LIN {X 0,Y 199.613,Z 290.431,A -85,B 0,C 180,E1 -21475.713,E2 -21475.713} C_VEL
LIN {X 0,Y 199.653,Z 290.436,A -85,B 0,C 180,E1 -21477.571,E2 -21477.571} C_VEL
LIN {X 0,Y 200.584,Z 293.129,A -85,B 0,C 180,E1 -21477.855,E2 -21477.855} C_VEL
LIN {X 0,Y 203.702,Z 298.377,A -85,B 0,C 180,E1 -21478.627,E2 -21478.627} C_VEL
LIN {X 0,Y 211.896,Z 314.5,A -85,B 0,C 180,E1 -21480.608,E2 -21480.608} C_VEL
LIN {X 0,Y 215.116,Z 321.856,A -85,B 0,C 180,E1 -21481.374,E2 -21481.374} C_VEL
LIN {X 0,Y 213.786,Z 358.585,A -85,B 0,C 180,E1 -21482.597,E2 -21482.597} C_VEL
LIN {X 0,Y 213.285,Z 367.836,A -85,B 0,C 180,E1 -21483.118,E2 -21483.118} C_VEL
LIN {X 0,Y 212.677,Z 375.597,A -85,B 0,C 180,E1 -21483.748,E2 -21483.748} C_VEL
LIN {X 0,Y 211.647,Z 384.419,A -85,B 0,C 180,E1 -21484.688,E2 -21484.688} C_VEL
LIN {X 0,Y 210.204,Z 392.837,A -85,B 0,C 180,E1 -21485.821,E2 -21485.821} C_VEL
LIN {X 0,Y 208.91,Z 399.701,A -85,B 0,C 180,E1 -21486.977,E2 -21486.977} C_VEL
LIN {X 0,Y 207.269,Z 407.588,A -85,B 0,C 180,E1 -21488.622,E2 -21488.622} C_VEL
LIN {X 0,Y 205.97,Z 413.247,A -85,B 0,C 180,E1 -21490.048,E2 -21490.048} C_VEL
LIN {X 0,Y 204.385,Z 419.566,A -85,B 0,C 180,E1 -21491.971,E2 -21491.971} C_VEL
LIN {X 0,Y 202.851,Z 424.822,A -85,B 0,C 180,E1 -21493.908,E2 -21493.908} C_VEL
LIN {X 0,Y 201.567,Z 429.206,A -85,B 0,C 180,E1 -21495.872,E2 -21495.872} C_VEL
LIN {X 0,Y 200.108,Z 434.351,A -85,B 0,C 180,E1 -21498.861,E2 -21498.861} C_VEL
LIN {X 0,Y 199.427,Z 436.755,A -85,B 0,C 180,E1 -21500.664,E2 -21500.664} C_VEL
LIN {X 0,Y 198.499,Z 439.877,A -85,B 0,C 180,E1 -21503.902,E2 -21503.902} C_VEL
LIN {X 0,Y 198.087,Z 441.139,A -85,B 0,C 180,E1 -21505.93,E2 -21505.93} C_VEL
LIN {X 0,Y 197.808,Z 441.935,A -85,B 0,C 180,E1 -21507.963,E2 -21507.963} C_VEL
LIN {X 0,Y 197.72,Z 442.238,A -85,B 0,C 180,E1 -21509.999,E2 -21509.999} C_VEL
LIN {X 0,Y 197.805,Z 441.958,A -85,B 0,C 180,E1 -21512.035,E2 -21512.035} C_VEL
LIN {X 0,Y 198.078,Z 441.21,A -85,B 0,C 180,E1 -21514.068,E2 -21514.068} C_VEL
LIN {X 0,Y 198.49,Z 439.996,A -85,B 0,C 180,E1 -21516.096,E2 -21516.096} C_VEL
LIN {X 0,Y 199.036,Z 438.296,A -85,B 0,C 180,E1 -21518.119,E2 -21518.119} C_VEL
LIN {X 0,Y 200.093,Z 434.572,A -85,B 0,C 180,E1 -21521.137,E2 -21521.137} C_VEL
LIN {X 0,Y 201.547,Z 429.487,A -85,B 0,C 180,E1 -21524.127,E2 -21524.127} C_VEL
LIN {X 0,Y 203.159,Z 424.005,A -85,B 0,C 180,E1 -21526.581,E2 -21526.581} C_VEL
LIN {X 0,Y 205.084,Z 417.109,A -85,B 0,C 180,E1 -21528.998,E2 -21528.998} C_VEL
LIN {X 0,Y 206.999,Z 409.189,A -85,B 0,C 180,E1 -21531.144,E2 -21531.144} C_VEL
LIN {X 0,Y 208.645,Z 401.633,A -85,B 0,C 180,E1 -21532.79,E2 -21532.79} C_VEL
LIN {X 0,Y 210.207,Z 393.703,A -85,B 0,C 180,E1 -21534.176,E2 -21534.176} C_VEL
LIN {X 0,Y 211.587,Z 385.502,A -85,B 0,C 180,E1 -21535.317,E2 -21535.317} C_VEL
LIN {X 0,Y 212.67,Z 377.081,A -85,B 0,C 180,E1 -21536.241,E2 -21536.241} C_VEL
LIN {X 0,Y 213.409,Z 367.929,A -85,B 0,C 180,E1 -21537.009,E2 -21537.009} C_VEL
LIN {X 0,Y 213.899,Z 358.992,A -85,B 0,C 180,E1 -21537.518,E2 -21537.518} C_VEL
LIN {X 0,Y 215.253,Z 322.206,A -85,B 0,C 180,E1 -21538.745,E2 -21538.745} C_VEL
LIN {X 0,Y 209.18,Z 308.863,A -85,B 0,C 180,E1 -21540.195,E2 -21540.195} C_VEL
LIN {X 0,Y 201.446,Z 294.316,A -85,B 0,C 180,E1 -21542.103,E2 -21542.103} C_VEL
LIN {X 0,Y 199.955,Z 291.746,A -85,B 0,C 180,E1 -21542.483,E2 -21542.483} C_VEL
LIN {X 0,Y 199.655,Z 290.429,A -85,B 0,C 180,E1 -21542.638,E2 -21542.638} C_VEL
LIN {X 0,Y 199.613,Z 290.425,A -85,B 0,C 180,E1 -21546.764,E2 -21546.764} C_VEL
LIN {X 0,Y 199.591,Z 290.435,A -85,B 0,C 180,E1 -21549.331,E2 -21549.331} C_VEL
LIN {X 0,Y 199.562,Z 290.428,A -85,B 0,C 180,E1 -21552.306,E2 -21552.306} C_VEL
LIN {X 0,Y 199.573,Z 290.436,A -85,B 0,C 180,E1 -21555.226,E2 -21555.226} C_VEL
LIN {X 0,Y 199.566,Z 290.42,A -85,B 0,C 180,E1 -21558.001,E2 -21558.001} C_VEL
LIN {X 0,Y 199.593,Z 290.431,A -85,B 0,C 180,E1 -21560.772,E2 -21560.772} C_VEL
LIN {X 0,Y 199.607,Z 290.432,A -85,B 0,C 180,E1 -21565.712,E2 -21565.712} C_VEL
LIN {X 0,Y 199.682,Z 290.419,A -85,B 0,C 180,E1 -21568.133,E2 -21568.133} C_VEL
LIN {X 0,Y 199.638,Z 290.422,A -85,B 0,C 180,E1 -21572.764,E2 -21572.764} C_VEL
LIN {X 0,Y 199.674,Z 290.421,A -85,B 0,C 180,E1 -21577.221,E2 -21577.221} C_VEL
LIN {X 0,Y 199.742,Z 290.411,A -85,B 0,C 180,E1 -21581.802,E2 -21581.802} C_VEL
LIN {X 0,Y 199.766,Z 290.389,A -85,B 0,C 180,E1 -21585.743,E2 -21585.743} C_VEL
LIN {X 0,Y 200.019,Z 290.381,A -85,B 0,C 180,E1 -21589.881,E2 -21589.881} C_VEL
LIN {X 0,Y 199.994,Z 290.372,A -85,B 0,C 180,E1 -21593.948,E2 -21593.948} C_VEL
LIN {X 0,Y 200.28,Z 290.332,A -85,B 0,C 180,E1 -21597.989,E2 -21597.989} C_VEL
LIN {X 0,Y 200.442,Z 290.324,A -85,B 0,C 180,E1 -21600,E2 -21600} C_VEL
LIN {X 0,Y 199.983,Z 290.383,A -85,B 0,C 180,E1 -21604.03,E2 -21604.03} C_VEL
LIN {X 0,Y 200.07,Z 290.377,A -85,B 0,C 180,E1 -21608.077,E2 -21608.077} C_VEL
LIN {X 0,Y 199.848,Z 290.402,A -85,B 0,C 180,E1 -21612.181,E2 -21612.181} C_VEL
LIN {X 0,Y 199.738,Z 290.415,A -85,B 0,C 180,E1 -21616.349,E2 -21616.349} C_VEL
LIN {X 0,Y 199.639,Z 290.427,A -85,B 0,C 180,E1 -21620.612,E2 -21620.612} C_VEL
LIN {X 0,Y 199.621,Z 290.428,A -85,B 0,C 180,E1 -21624.991,E2 -21624.991} C_VEL
LIN {X 0,Y 199.602,Z 290.437,A -85,B 0,C 180,E1 -21629.534,E2 -21629.534} C_VEL
LIN {X 0,Y 199.661,Z 290.429,A -85,B 0,C 180,E1 -21632.353,E2 -21632.353} C_VEL
LIN {X 0,Y 199.611,Z 290.436,A -85,B 0,C 180,E1 -21636.765,E2 -21636.765} C_VEL
LIN {X 0,Y 199.59,Z 290.44,A -85,B 0,C 180,E1 -21639.332,E2 -21639.332} C_VEL
LIN {X 0,Y 199.561,Z 290.441,A -85,B 0,C 180,E1 -21642.308,E2 -21642.308} C_VEL
LIN {X 0,Y 199.572,Z 290.441,A -85,B 0,C 180,E1 -21645.228,E2 -21645.228} C_VEL
LIN {X 0,Y 199.566,Z 290.44,A -85,B 0,C 180,E1 -21648.003,E2 -21648.003} C_VEL
LIN {X 0,Y 199.653,Z 290.544,A -85,B 0,C 180,E1 -21651.413,E2 -21651.413} C_VEL
LIN {X 0,Y 201.4,Z 297.896,A -85,B 0,C 180,E1 -21655.456,E2 -21655.456} C_VEL
LIN {X 0,Y 202.273,Z 302.073,A -85,B 0,C 180,E1 -21657.631,E2 -21657.631} C_VEL
LIN {X 0,Y 208.961,Z 318.344,A -85,B 0,C 180,E1 -21659.408,E2 -21659.408} C_VEL
LIN {X 0,Y 210.715,Z 328.85,A -85,B 0,C 180,E1 -21660.089,E2 -21660.089} C_VEL
LIN {X 0,Y 211.052,Z 334.648,A -85,B 0,C 180,E1 -21660.363,E2 -21660.363} C_VEL
LIN {X 0,Y 209.97,Z 344.437,A -85,B 0,C 180,E1 -21660.573,E2 -21660.573} C_VEL
LIN {X 0,Y 208.579,Z 352.327,A -85,B 0,C 180,E1 -21660.665,E2 -21660.665} C_VEL
LIN {X 0,Y 207.672,Z 360.248,A -85,B 0,C 180,E1 -21660.833,E2 -21660.833} C_VEL
LIN {X 0,Y 206.792,Z 381.239,A -85,B 0,C 180,E1 -21661.59,E2 -21661.59} C_VEL
LIN {X 0,Y 205.784,Z 392.316,A -85,B 0,C 180,E1 -21662.27,E2 -21662.27} C_VEL
LIN {X 0,Y 204.008,Z 403.947,A -85,B 0,C 180,E1 -21663.396,E2 -21663.396} C_VEL
LIN {X 0,Y 202.279,Z 413.34,A -85,B 0,C 180,E1 -21664.666,E2 -21664.666} C_VEL
LIN {X 0,Y 200.62,Z 420.935,A -85,B 0,C 180,E1 -21665.97,E2 -21665.97} C_VEL
LIN {X 0,Y 198.696,Z 428.802,A -85,B 0,C 180,E1 -21667.653,E2 -21667.653} C_VEL
LIN {X 0,Y 196.738,Z 436.167,A -85,B 0,C 180,E1 -21669.618,E2 -21669.618} C_VEL
LIN {X 0,Y 194.702,Z 443.648,A -85,B 0,C 180,E1 -21672.134,E2 -21672.134} C_VEL
LIN {X 0,Y 192.709,Z 450.484,A -85,B 0,C 180,E1 -21675.211,E2 -21675.211} C_VEL
LIN {X 0,Y 191.391,Z 455.696,A -85,B 0,C 180,E1 -21678.349,E2 -21678.349} C_VEL
LIN {X 0,Y 190.642,Z 459.536,A -85,B 0,C 180,E1 -21681.521,E2 -21681.521} C_VEL
LIN {X 0,Y 190.376,Z 461.305,A -85,B 0,C 180,E1 -21683.643,E2 -21683.643} C_VEL
LIN {X 0,Y 190.315,Z 462.576,A -85,B 0,C 180,E1 -21685.766,E2 -21685.766} C_VEL
LIN {X 0,Y 190.441,Z 463.373,A -85,B 0,C 180,E1 -21687.886,E2 -21687.886} C_VEL
LIN {X 0,Y 190.608,Z 463.679,A -85,B 0,C 180,E1 -21690.001,E2 -21690.001} C_VEL
LIN {X 0,Y 190.444,Z 463.364,A -85,B 0,C 180,E1 -21692.116,E2 -21692.116} C_VEL
LIN {X 0,Y 190.335,Z 462.437,A -85,B 0,C 180,E1 -21694.474,E2 -21694.474} C_VEL
LIN {X 0,Y 190.378,Z 461.256,A -85,B 0,C 180,E1 -21696.36,E2 -21696.36} C_VEL
LIN {X 0,Y 190.856,Z 458.298,A -85,B 0,C 180,E1 -21699.539,E2 -21699.539} C_VEL
LIN {X 0,Y 191.391,Z 455.606,A -85,B 0,C 180,E1 -21701.653,E2 -21701.653} C_VEL
LIN {X 0,Y 192.708,Z 450.367,A -85,B 0,C 180,E1 -21704.792,E2 -21704.792} C_VEL
LIN {X 0,Y 194.692,Z 443.478,A -85,B 0,C 180,E1 -21707.87,E2 -21707.87} C_VEL
LIN {X 0,Y 196.719,Z 435.963,A -85,B 0,C 180,E1 -21710.386,E2 -21710.386} C_VEL
LIN {X 0,Y 198.719,Z 428.564,A -85,B 0,C 180,E1 -21712.347,E2 -21712.347} C_VEL
LIN {X 0,Y 200.645,Z 420.642,A -85,B 0,C 180,E1 -21714.029,E2 -21714.029} C_VEL
LIN {X 0,Y 202.677,Z 410.766,A -85,B 0,C 180,E1 -21715.686,E2 -21715.686} C_VEL
LIN {X 0,Y 204.651,Z 399.203,A -85,B 0,C 180,E1 -21717.067,E2 -21717.067} C_VEL
LIN {X 0,Y 205.966,Z 389.853,A -85,B 0,C 180,E1 -21717.844,E2 -21717.844} C_VEL
LIN {X 0,Y 206.816,Z 379.973,A -85,B 0,C 180,E1 -21718.409,E2 -21718.409} C_VEL
LIN {X 0,Y 207.545,Z 357.654,A -85,B 0,C 180,E1 -21719.221,E2 -21719.221} C_VEL
LIN {X 0,Y 205.525,Z 338.227,A -85,B 0,C 180,E1 -21720.295,E2 -21720.295} C_VEL
LIN {X 0,Y 203.229,Z 321.421,A -85,B 0,C 180,E1 -21721.343,E2 -21721.343} C_VEL
LIN {X 0,Y 197.805,Z 308.229,A -85,B 0,C 180,E1 -21722.844,E2 -21722.844} C_VEL
LIN {X 0,Y 194.959,Z 301.496,A -85,B 0,C 180,E1 -21723.721,E2 -21723.721} C_VEL
LIN {X 0,Y 193.277,Z 294.173,A -85,B 0,C 180,E1 -21727.825,E2 -21727.825} C_VEL
LIN {X 0,Y 192.543,Z 291.315,A -85,B 0,C 180,E1 -21729.562,E2 -21729.562} C_VEL
LIN {X 0,Y 192.488,Z 291.323,A -85,B 0,C 180,E1 -21733.926,E2 -21733.926} C_VEL
LIN {X 0,Y 192.505,Z 291.321,A -85,B 0,C 180,E1 -21738.918,E2 -21738.918} C_VEL
LIN {X 0,Y 192.582,Z 291.31,A -85,B 0,C 180,E1 -21743.405,E2 -21743.405} C_VEL
LIN {X 0,Y 192.607,Z 291.306,A -85,B 0,C 180,E1 -21747.062,E2 -21747.062} C_VEL
LIN {X 0,Y 192.613,Z 291.303,A -85,B 0,C 180,E1 -21751.684,E2 -21751.684} C_VEL
LIN {X 0,Y 192.658,Z 291.298,A -85,B 0,C 180,E1 -21756.343,E2 -21756.343} C_VEL
LIN {X 0,Y 192.697,Z 291.294,A -85,B 0,C 180,E1 -21761.492,E2 -21761.492} C_VEL
LIN {X 0,Y 192.775,Z 291.285,A -85,B 0,C 180,E1 -21767.365,E2 -21767.365} C_VEL
LIN {X 0,Y 193.021,Z 291.223,A -85,B 0,C 180,E1 -21771.626,E2 -21771.626} C_VEL
LIN {X 0,Y 193.229,Z 291.228,A -85,B 0,C 180,E1 -21777.916,E2 -21777.916} C_VEL
LIN {X 0,Y 193.416,Z 291.198,A -85,B 0,C 180,E1 -21780,E2 -21780} C_VEL
LIN {X 0,Y 192.933,Z 291.235,A -85,B 0,C 180,E1 -21784.178,E2 -21784.178} C_VEL
LIN {X 0,Y 193.024,Z 291.251,A -85,B 0,C 180,E1 -21788.375,E2 -21788.375} C_VEL
LIN {X 0,Y 192.778,Z 291.27,A -85,B 0,C 180,E1 -21792.635,E2 -21792.635} C_VEL
LIN {X 0,Y 192.697,Z 291.288,A -85,B 0,C 180,E1 -21798.508,E2 -21798.508} C_VEL
LIN {X 0,Y 192.613,Z 291.3,A -85,B 0,C 180,E1 -21804.188,E2 -21804.188} C_VEL
LIN {X 0,Y 192.603,Z 291.302,A -85,B 0,C 180,E1 -21808.864,E2 -21808.864} C_VEL
LIN {X 0,Y 192.597,Z 291.295,A -85,B 0,C 180,E1 -21813.186,E2 -21813.186} C_VEL
LIN {X 0,Y 192.543,Z 291.314,A -85,B 0,C 180,E1 -21818.354,E2 -21818.354} C_VEL
LIN {X 0,Y 192.485,Z 291.307,A -85,B 0,C 180,E1 -21823.092,E2 -21823.092} C_VEL
LIN {X 0,Y 192.487,Z 291.323,A -85,B 0,C 180,E1 -21826.906,E2 -21826.906} C_VEL
LIN {X 0,Y 192.543,Z 291.267,A -85,B 0,C 180,E1 -21831.645,E2 -21831.645} C_VEL
LIN {X 0,Y 192.602,Z 291.389,A -85,B 0,C 180,E1 -21836.249,E2 -21836.249} C_VEL
LIN {X 0,Y 193.654,Z 294.262,A -85,B 0,C 180,E1 -21836.586,E2 -21836.586} C_VEL
LIN {X 0,Y 195.306,Z 296.896,A -85,B 0,C 180,E1 -21837.023,E2 -21837.023} C_VEL
LIN {X 0,Y 201.653,Z 308.403,A -85,B 0,C 180,E1 -21838.677,E2 -21838.677} C_VEL
LIN {X 0,Y 208.096,Z 321.908,A -85,B 0,C 180,E1 -21840.297,E2 -21840.297} C_VEL
LIN {X 0,Y 208.918,Z 323.896,A -85,B 0,C 180,E1 -21840.505,E2 -21840.505} C_VEL
LIN {X 0,Y 207.509,Z 359.706,A -85,B 0,C 180,E1 -21841.733,E2 -21841.733} C_VEL
LIN {X 0,Y 206.913,Z 368.837,A -85,B 0,C 180,E1 -21842.269,E2 -21842.269} C_VEL
LIN {X 0,Y 206.141,Z 378.024,A -85,B 0,C 180,E1 -21843.079,E2 -21843.079} C_VEL
LIN {X 0,Y 204.99,Z 386.681,A -85,B 0,C 180,E1 -21844.078,E2 -21844.078} C_VEL
LIN {X 0,Y 203.197,Z 396.224,A -85,B 0,C 180,E1 -21845.477,E2 -21845.477} C_VEL
LIN {X 0,Y 201.461,Z 404.915,A -85,B 0,C 180,E1 -21847.163,E2 -21847.163} C_VEL
LIN {X 0,Y 199.341,Z 413.64,A -85,B 0,C 180,E1 -21849.355,E2 -21849.355} C_VEL
LIN {X 0,Y 197.667,Z 419.959,A -85,B 0,C 180,E1 -21851.337,E2 -21851.337} C_VEL
LIN {X 0,Y 196.071,Z 425.215,A -85,B 0,C 180,E1 -21853.335,E2 -21853.335} C_VEL
LIN {X 0,Y 194.71,Z 429.598,A -85,B 0,C 180,E1 -21855.364,E2 -21855.364} C_VEL
LIN {X 0,Y 193.159,Z 434.744,A -85,B 0,C 180,E1 -21858.455,E2 -21858.455} C_VEL
LIN {X 0,Y 192.374,Z 437.381,A -85,B 0,C 180,E1 -21860.538,E2 -21860.538} C_VEL
LIN {X 0,Y 191.458,Z 440.269,A -85,B 0,C 180,E1 -21863.677,E2 -21863.677} C_VEL
LIN {X 0,Y 191.042,Z 441.529,A -85,B 0,C 180,E1 -21865.78,E2 -21865.78} C_VEL
LIN {X 0,Y 190.748,Z 442.325,A -85,B 0,C 180,E1 -21867.887,E2 -21867.887} C_VEL
LIN {X 0,Y 190.655,Z 442.628,A -85,B 0,C 180,E1 -21869.999,E2 -21869.999} C_VEL
LIN {X 0,Y 190.745,Z 442.348,A -85,B 0,C 180,E1 -21872.11,E2 -21872.11} C_VEL
LIN {X 0,Y 191.034,Z 441.599,A -85,B 0,C 180,E1 -21874.218,E2 -21874.218} C_VEL
LIN {X 0,Y 191.449,Z 440.387,A -85,B 0,C 180,E1 -21876.322,E2 -21876.322} C_VEL
LIN {X 0,Y 192.316,Z 437.661,A -85,B 0,C 180,E1 -21879.358,E2 -21879.358} C_VEL
LIN {X 0,Y 193.151,Z 434.962,A -85,B 0,C 180,E1 -21881.543,E2 -21881.543} C_VEL
LIN {X 0,Y 194.69,Z 429.876,A -85,B 0,C 180,E1 -21884.636,E2 -21884.636} C_VEL
LIN {X 0,Y 196.377,Z 424.395,A -85,B 0,C 180,E1 -21887.172,E2 -21887.172} C_VEL
LIN {X 0,Y 198.419,Z 417.496,A -85,B 0,C 180,E1 -21889.662,E2 -21889.662} C_VEL
LIN {X 0,Y 200.402,Z 409.577,A -85,B 0,C 180,E1 -21891.876,E2 -21891.876} C_VEL
LIN {X 0,Y 202.139,Z 402.02,A -85,B 0,C 180,E1 -21893.567,E2 -21893.567} C_VEL
LIN {X 0,Y 203.786,Z 394.088,A -85,B 0,C 180,E1 -21894.989,E2 -21894.989} C_VEL
LIN {X 0,Y 205.222,Z 385.886,A -85,B 0,C 180,E1 -21896.161,E2 -21896.161} C_VEL
LIN {X 0,Y 206.312,Z 377.646,A -85,B 0,C 180,E1 -21897.094,E2 -21897.094} C_VEL
LIN {X 0,Y 207.096,Z 368.746,A -85,B 0,C 180,E1 -21897.866,E2 -21897.866} C_VEL
LIN {X 0,Y 207.647,Z 359.505,A -85,B 0,C 180,E1 -21898.413,E2 -21898.413} C_VEL
LIN {X 0,Y 209.064,Z 324.183,A -85,B 0,C 180,E1 -21899.617,E2 -21899.617} C_VEL
LIN {X 0,Y 202.494,Z 310.086,A -85,B 0,C 180,E1 -21901.269,E2 -21901.269} C_VEL
LIN {X 0,Y 196.233,Z 298.469,A -85,B 0,C 180,E1 -21902.899,E2 -21902.899} C_VEL
LIN {X 0,Y 194.061,Z 294.841,A -85,B 0,C 180,E1 -21903.479,E2 -21903.479} C_VEL
LIN {X 0,Y 192.734,Z 292.117,A -85,B 0,C 180,E1 -21903.864,E2 -21903.864} C_VEL
LIN {X 0,Y 192.573,Z 291.311,A -85,B 0,C 180,E1 -21903.954,E2 -21903.954} C_VEL
LIN {X 0,Y 192.538,Z 291.315,A -85,B 0,C 180,E1 -21908.353,E2 -21908.353} C_VEL
LIN {X 0,Y 192.482,Z 291.316,A -85,B 0,C 180,E1 -21913.092,E2 -21913.092} C_VEL
LIN {X 0,Y 192.481,Z 291.306,A -85,B 0,C 180,E1 -21916.906,E2 -21916.906} C_VEL
LIN {X 0,Y 192.537,Z 291.313,A -85,B 0,C 180,E1 -21921.645,E2 -21921.645} C_VEL
LIN {X 0,Y 192.591,Z 291.303,A -85,B 0,C 180,E1 -21926.812,E2 -21926.812} C_VEL
LIN {X 0,Y 192.616,Z 291.298,A -85,B 0,C 180,E1 -21931.684,E2 -21931.684} C_VEL
LIN {X 0,Y 192.667,Z 291.295,A -85,B 0,C 180,E1 -21936.343,E2 -21936.343} C_VEL
LIN {X 0,Y 192.69,Z 291.291,A -85,B 0,C 180,E1 -21941.491,E2 -21941.491} C_VEL
LIN {X 0,Y 192.77,Z 291.27,A -85,B 0,C 180,E1 -21947.364,E2 -21947.364} C_VEL
LIN {X 0,Y 193.017,Z 291.252,A -85,B 0,C 180,E1 -21951.625,E2 -21951.625} C_VEL
LIN {X 0,Y 193.224,Z 291.208,A -85,B 0,C 180,E1 -21957.915,E2 -21957.915} C_VEL
LIN {X 0,Y 193.409,Z 291.199,A -85,B 0,C 180,E1 -21960,E2 -21960} C_VEL
LIN {X 0,Y 192.93,Z 291.26,A -85,B 0,C 180,E1 -21964.178,E2 -21964.178} C_VEL
LIN {X 0,Y 193.021,Z 291.254,A -85,B 0,C 180,E1 -21968.374,E2 -21968.374} C_VEL
LIN {X 0,Y 192.77,Z 291.286,A -85,B 0,C 180,E1 -21972.635,E2 -21972.635} C_VEL
LIN {X 0,Y 192.69,Z 291.295,A -85,B 0,C 180,E1 -21978.508,E2 -21978.508} C_VEL
LIN {X 0,Y 192.616,Z 291.301,A -85,B 0,C 180,E1 -21984.195,E2 -21984.195} C_VEL
LIN {X 0,Y 192.596,Z 291.309,A -85,B 0,C 180,E1 -21988.865,E2 -21988.865} C_VEL
LIN {X 0,Y 192.59,Z 291.311,A -85,B 0,C 180,E1 -21993.187,E2 -21993.187} C_VEL
LIN {X 0,Y 192.536,Z 291.317,A -85,B 0,C 180,E1 -21998.355,E2 -21998.355} C_VEL
LIN {X 0,Y 192.481,Z 291.325,A -85,B 0,C 180,E1 -22003.094,E2 -22003.094} C_VEL
LIN {X 0,Y 192.481,Z 291.324,A -85,B 0,C 180,E1 -22006.907,E2 -22006.907} C_VEL
LIN {X 0,Y 192.57,Z 291.456,A -85,B 0,C 180,E1 -22010.485,E2 -22010.485} C_VEL
LIN {X 0,Y 194.337,Z 298.658,A -85,B 0,C 180,E1 -22014.648,E2 -22014.648} C_VEL
LIN {X 0,Y 194.997,Z 301.675,A -85,B 0,C 180,E1 -22016.27,E2 -22016.27} C_VEL
LIN {X 0,Y 201.837,Z 317.661,A -85,B 0,C 180,E1 -22018.194,E2 -22018.194} C_VEL
LIN {X 0,Y 203.421,Z 322.25,A -85,B 0,C 180,E1 -22018.652,E2 -22018.652} C_VEL
LIN {X 0,Y 206.196,Z 342.981,A -85,B 0,C 180,E1 -22019.932,E2 -22019.932} C_VEL
LIN {X 0,Y 207.732,Z 358.961,A -85,B 0,C 180,E1 -22020.793,E2 -22020.793} C_VEL
LIN {X 0,Y 207.672,Z 360.248,A -85,B 0,C 180,E1 -22020.833,E2 -22020.833} C_VEL
LIN {X 0,Y 206.824,Z 366.093,A -85,B 0,C 180,E1 -22020.918,E2 -22020.918} C_VEL
LIN {X 0,Y 201.247,Z 383.078,A -85,B 0,C 180,E1 -22020.852,E2 -22020.852} C_VEL
LIN {X 0,Y 200.271,Z 386.871,A -85,B 0,C 180,E1 -22020.997,E2 -22020.997} C_VEL
LIN {X 0,Y 199.662,Z 390.687,A -85,B 0,C 180,E1 -22021.234,E2 -22021.234} C_VEL
LIN {X 0,Y 198.038,Z 401.668,A -85,B 0,C 180,E1 -22022.241,E2 -22022.241} C_VEL
LIN {X 0,Y 196.121,Z 411.756,A -85,B 0,C 180,E1 -22023.584,E2 -22023.584} C_VEL
LIN {X 0,Y 194.418,Z 419.334,A -85,B 0,C 180,E1 -22024.872,E2 -22024.872} C_VEL
LIN {X 0,Y 192.427,Z 427.389,A -85,B 0,C 180,E1 -22026.599,E2 -22026.599} C_VEL
LIN {X 0,Y 190.541,Z 434.062,A -85,B 0,C 180,E1 -22028.357,E2 -22028.357} C_VEL
LIN {X 0,Y 188.772,Z 440.411,A -85,B 0,C 180,E1 -22030.424,E2 -22030.424} C_VEL
LIN {X 0,Y 187.155,Z 445.686,A -85,B 0,C 180,E1 -22032.519,E2 -22032.519} C_VEL
LIN {X 0,Y 185.821,Z 450.091,A -85,B 0,C 180,E1 -22034.649,E2 -22034.649} C_VEL
LIN {X 0,Y 184.416,Z 455.304,A -85,B 0,C 180,E1 -22037.902,E2 -22037.902} C_VEL
LIN {X 0,Y 183.597,Z 459.144,A -85,B 0,C 180,E1 -22041.194,E2 -22041.194} C_VEL
LIN {X 0,Y 183.31,Z 460.913,A -85,B 0,C 180,E1 -22043.396,E2 -22043.396} C_VEL
LIN {X 0,Y 183.232,Z 462.25,A -85,B 0,C 180,E1 -22045.748,E2 -22045.748} C_VEL
LIN {X 0,Y 183.354,Z 462.982,A -85,B 0,C 180,E1 -22047.804,E2 -22047.804} C_VEL
LIN {X 0,Y 183.54,Z 463.289,A -85,B 0,C 180,E1 -22050.001,E2 -22050.001} C_VEL
LIN {X 0,Y 183.357,Z 462.972,A -85,B 0,C 180,E1 -22052.198,E2 -22052.198} C_VEL
LIN {X 0,Y 183.236,Z 462.155,A -85,B 0,C 180,E1 -22054.401,E2 -22054.401} C_VEL
LIN {X 0,Y 183.311,Z 460.863,A -85,B 0,C 180,E1 -22056.606,E2 -22056.606} C_VEL
LIN {X 0,Y 183.828,Z 457.903,A -85,B 0,C 180,E1 -22059.908,E2 -22059.908} C_VEL
LIN {X 0,Y 184.417,Z 455.211,A -85,B 0,C 180,E1 -22062.1,E2 -22062.1} C_VEL
LIN {X 0,Y 185.82,Z 449.972,A -85,B 0,C 180,E1 -22065.353,E2 -22065.353} C_VEL
LIN {X 0,Y 187.906,Z 443.082,A -85,B 0,C 180,E1 -22068.538,E2 -22068.538} C_VEL
LIN {X 0,Y 190.045,Z 435.566,A -85,B 0,C 180,E1 -22071.136,E2 -22071.136} C_VEL
LIN {X 0,Y 192.184,Z 428.169,A -85,B 0,C 180,E1 -22073.15,E2 -22073.15} C_VEL
LIN {X 0,Y 194.156,Z 420.29,A -85,B 0,C 180,E1 -22074.876,E2 -22074.876} C_VEL
LIN {X 0,Y 196.002,Z 411.76,A -85,B 0,C 180,E1 -22076.364,E2 -22076.364} C_VEL
LIN {X 0,Y 198.012,Z 401.156,A -85,B 0,C 180,E1 -22077.766,E2 -22077.766} C_VEL
LIN {X 0,Y 199.635,Z 390.284,A -85,B 0,C 180,E1 -22078.736,E2 -22078.736} C_VEL
LIN {X 0,Y 200.517,Z 380.864,A -85,B 0,C 180,E1 -22079.315,E2 -22079.315} C_VEL
LIN {X 0,Y 201.341,Z 358.404,A -85,B 0,C 180,E1 -22080.166,E2 -22080.166} C_VEL
LIN {X 0,Y 198.962,Z 335.352,A -85,B 0,C 180,E1 -22081.506,E2 -22081.506} C_VEL
LIN {X 0,Y 197.161,Z 323.377,A -85,B 0,C 180,E1 -22082.324,E2 -22082.324} C_VEL
LIN {X 0,Y 191.451,Z 309.451,A -85,B 0,C 180,E1 -22084.007,E2 -22084.007} C_VEL
LIN {X 0,Y 187.63,Z 300.989,A -85,B 0,C 180,E1 -22085.238,E2 -22085.238} C_VEL
LIN {X 0,Y 186.078,Z 294.602,A -85,B 0,C 180,E1 -22089.041,E2 -22089.041} C_VEL
LIN {X 0,Y 185.466,Z 292.197,A -85,B 0,C 180,E1 -22090.63,E2 -22090.63} C_VEL
LIN {X 0,Y 185.456,Z 292.199,A -85,B 0,C 180,E1 -22096.057,E2 -22096.057} C_VEL
LIN {X 0,Y 185.457,Z 292.199,A -85,B 0,C 180,E1 -22099.893,E2 -22099.893} C_VEL
LIN {X 0,Y 185.502,Z 292.195,A -85,B 0,C 180,E1 -22102.715,E2 -22102.715} C_VEL
LIN {X 0,Y 185.532,Z 292.186,A -85,B 0,C 180,E1 -22107.973,E2 -22107.973} C_VEL
LIN {X 0,Y 185.494,Z 292.193,A -85,B 0,C 180,E1 -22112.957,E2 -22112.957} C_VEL
LIN {X 0,Y 185.547,Z 292.186,A -85,B 0,C 180,E1 -22117.743,E2 -22117.743} C_VEL
LIN {X 0,Y 185.648,Z 292.172,A -85,B 0,C 180,E1 -22122.371,E2 -22122.371} C_VEL
LIN {X 0,Y 185.699,Z 292.165,A -85,B 0,C 180,E1 -22126.875,E2 -22126.875} C_VEL
LIN {X 0,Y 185.972,Z 292.101,A -85,B 0,C 180,E1 -22131.306,E2 -22131.306} C_VEL
LIN {X 0,Y 186.175,Z 292.107,A -85,B 0,C 180,E1 -22137.837,E2 -22137.837} C_VEL
LIN {X 0,Y 186.381,Z 292.074,A -85,B 0,C 180,E1 -22140,E2 -22140} C_VEL
LIN {X 0,Y 185.881,Z 292.112,A -85,B 0,C 180,E1 -22144.337,E2 -22144.337} C_VEL
LIN {X 0,Y 185.975,Z 292.13,A -85,B 0,C 180,E1 -22148.694,E2 -22148.694} C_VEL
LIN {X 0,Y 185.701,Z 292.147,A -85,B 0,C 180,E1 -22153.125,E2 -22153.125} C_VEL
LIN {X 0,Y 185.628,Z 292.17,A -85,B 0,C 180,E1 -22158.821,E2 -22158.821} C_VEL
LIN {X 0,Y 185.547,Z 292.183,A -85,B 0,C 180,E1 -22164.623,E2 -22164.623} C_VEL
LIN {X 0,Y 185.546,Z 292.183,A -85,B 0,C 180,E1 -22169.499,E2 -22169.499} C_VEL
LIN {X 0,Y 185.499,Z 292.169,A -85,B 0,C 180,E1 -22174.632,E2 -22174.632} C_VEL
LIN {X 0,Y 185.502,Z 292.186,A -85,B 0,C 180,E1 -22177.314,E2 -22177.314} C_VEL
LIN {X 0,Y 185.462,Z 292.191,A -85,B 0,C 180,E1 -22180.72,E2 -22180.72} C_VEL
LIN {X 0,Y 185.458,Z 292.201,A -85,B 0,C 180,E1 -22186.056,E2 -22186.056} C_VEL
LIN {X 0,Y 185.457,Z 292.16,A -85,B 0,C 180,E1 -22189.891,E2 -22189.891} C_VEL
LIN {X 0,Y 185.533,Z 292.17,A -85,B 0,C 180,E1 -22194.775,E2 -22194.775} C_VEL
LIN {X 0,Y 186.508,Z 295.001,A -85,B 0,C 180,E1 -22195.136,E2 -22195.136} C_VEL
LIN {X 0,Y 187.868,Z 296.933,A -85,B 0,C 180,E1 -22195.517,E2 -22195.517} C_VEL
LIN {X 0,Y 195.088,Z 309.797,A -85,B 0,C 180,E1 -22197.537,E2 -22197.537} C_VEL
LIN {X 0,Y 201.924,Z 323.895,A -85,B 0,C 180,E1 -22199.357,E2 -22199.357} C_VEL
LIN {X 0,Y 202.733,Z 325.751,A -85,B 0,C 180,E1 -22199.57,E2 -22199.57} C_VEL
LIN {X 0,Y 201.341,Z 359.4,A -85,B 0,C 180,E1 -22200.745,E2 -22200.745} C_VEL
LIN {X 0,Y 200.752,Z 368.575,A -85,B 0,C 180,E1 -22201.284,E2 -22201.284} C_VEL
LIN {X 0,Y 200.014,Z 376.836,A -85,B 0,C 180,E1 -22201.997,E2 -22201.997} C_VEL
LIN {X 0,Y 198.953,Z 385.212,A -85,B 0,C 180,E1 -22202.946,E2 -22202.946} C_VEL
LIN {X 0,Y 197.404,Z 393.627,A -85,B 0,C 180,E1 -22204.142,E2 -22204.142} C_VEL
LIN {X 0,Y 195.716,Z 401.714,A -85,B 0,C 180,E1 -22205.608,E2 -22205.608} C_VEL
LIN {X 0,Y 193.923,Z 409.39,A -85,B 0,C 180,E1 -22207.351,E2 -22207.351} C_VEL
LIN {X 0,Y 191.803,Z 417.417,A -85,B 0,C 180,E1 -22209.628,E2 -22209.628} C_VEL
LIN {X 0,Y 189.696,Z 424.442,A -85,B 0,C 180,E1 -22212.202,E2 -22212.202} C_VEL
LIN {X 0,Y 187.859,Z 429.991,A -85,B 0,C 180,E1 -22214.817,E2 -22214.817} C_VEL
LIN {X 0,Y 186.218,Z 435.137,A -85,B 0,C 180,E1 -22218.019,E2 -22218.019} C_VEL
LIN {X 0,Y 185.257,Z 438.138,A -85,B 0,C 180,E1 -22220.523,E2 -22220.523} C_VEL
LIN {X 0,Y 184.423,Z 440.66,A -85,B 0,C 180,E1 -22223.434,E2 -22223.434} C_VEL
LIN {X 0,Y 184,Z 441.919,A -85,B 0,C 180,E1 -22225.618,E2 -22225.618} C_VEL
LIN {X 0,Y 183.69,Z 442.715,A -85,B 0,C 180,E1 -22227.806,E2 -22227.806} C_VEL
LIN {X 0,Y 183.591,Z 443.018,A -85,B 0,C 180,E1 -22229.999,E2 -22229.999} C_VEL
LIN {X 0,Y 183.687,Z 442.738,A -85,B 0,C 180,E1 -22232.192,E2 -22232.192} C_VEL
LIN {X 0,Y 183.969,Z 441.99,A -85,B 0,C 180,E1 -22234.381,E2 -22234.381} C_VEL
LIN {X 0,Y 184.414,Z 440.777,A -85,B 0,C 180,E1 -22236.564,E2 -22236.564} C_VEL
LIN {X 0,Y 185.239,Z 438.336,A -85,B 0,C 180,E1 -22239.444,E2 -22239.444} C_VEL
LIN {X 0,Y 186.212,Z 435.352,A -85,B 0,C 180,E1 -22241.979,E2 -22241.979} C_VEL
LIN {X 0,Y 187.836,Z 430.266,A -85,B 0,C 180,E1 -22245.182,E2 -22245.182} C_VEL
LIN {X 0,Y 189.631,Z 424.783,A -85,B 0,C 180,E1 -22247.802,E2 -22247.802} C_VEL
LIN {X 0,Y 191.776,Z 417.884,A -85,B 0,C 180,E1 -22250.373,E2 -22250.373} C_VEL
LIN {X 0,Y 193.834,Z 409.965,A -85,B 0,C 180,E1 -22252.657,E2 -22252.657} C_VEL
LIN {X 0,Y 195.665,Z 402.407,A -85,B 0,C 180,E1 -22254.396,E2 -22254.396} C_VEL
LIN {X 0,Y 197.407,Z 394.473,A -85,B 0,C 180,E1 -22255.855,E2 -22255.855} C_VEL
LIN {X 0,Y 198.89,Z 386.271,A -85,B 0,C 180,E1 -22257.06,E2 -22257.06} C_VEL
LIN {X 0,Y 200.01,Z 378.285,A -85,B 0,C 180,E1 -22257.991,E2 -22257.991} C_VEL
LIN {X 0,Y 200.863,Z 369.04,A -85,B 0,C 180,E1 -22258.818,E2 -22258.818} C_VEL
LIN {X 0,Y 201.464,Z 359.738,A -85,B 0,C 180,E1 -22259.377,E2 -22259.377} C_VEL
LIN {X 0,Y 202.794,Z 325.875,A -85,B 0,C 180,E1 -22260.576,E2 -22260.576} C_VEL
LIN {X 0,Y 195.729,Z 311.016,A -85,B 0,C 180,E1 -22262.457,E2 -22262.457} C_VEL
LIN {X 0,Y 189.3,Z 299.472,A -85,B 0,C 180,E1 -22264.241,E2 -22264.241} C_VEL
LIN {X 0,Y 187.072,Z 295.821,A -85,B 0,C 180,E1 -22264.881,E2 -22264.881} C_VEL
LIN {X 0,Y 185.687,Z 293.129,A -85,B 0,C 180,E1 -22265.309,E2 -22265.309} C_VEL
LIN {X 0,Y 185.504,Z 292.182,A -85,B 0,C 180,E1 -22265.396,E2 -22265.396} C_VEL
LIN {X 0,Y 185.458,Z 292.183,A -85,B 0,C 180,E1 -22270.719,E2 -22270.719} C_VEL
LIN {X 0,Y 185.452,Z 292.187,A -85,B 0,C 180,E1 -22276.056,E2 -22276.056} C_VEL
LIN {X 0,Y 185.452,Z 292.187,A -85,B 0,C 180,E1 -22279.891,E2 -22279.891} C_VEL
LIN {X 0,Y 185.497,Z 292.186,A -85,B 0,C 180,E1 -22282.713,E2 -22282.713} C_VEL
LIN {X 0,Y 185.527,Z 292.181,A -85,B 0,C 180,E1 -22287.971,E2 -22287.971} C_VEL
LIN {X 0,Y 185.544,Z 292.183,A -85,B 0,C 180,E1 -22290.595,E2 -22290.595} C_VEL
LIN {X 0,Y 185.577,Z 292.181,A -85,B 0,C 180,E1 -22295.381,E2 -22295.381} C_VEL
LIN {X 0,Y 185.621,Z 292.173,A -85,B 0,C 180,E1 -22301.178,E2 -22301.178} C_VEL
LIN {X 0,Y 185.694,Z 292.146,A -85,B 0,C 180,E1 -22306.874,E2 -22306.874} C_VEL
LIN {X 0,Y 185.968,Z 292.131,A -85,B 0,C 180,E1 -22311.305,E2 -22311.305} C_VEL
LIN {X 0,Y 186.17,Z 292.084,A -85,B 0,C 180,E1 -22317.836,E2 -22317.836} C_VEL
LIN {X 0,Y 186.375,Z 292.076,A -85,B 0,C 180,E1 -22320,E2 -22320} C_VEL
LIN {X 0,Y 185.878,Z 292.137,A -85,B 0,C 180,E1 -22324.337,E2 -22324.337} C_VEL
LIN {X 0,Y 185.97,Z 292.13,A -85,B 0,C 180,E1 -22328.694,E2 -22328.694} C_VEL
LIN {X 0,Y 185.694,Z 292.166,A -85,B 0,C 180,E1 -22333.125,E2 -22333.125} C_VEL
LIN {X 0,Y 185.621,Z 292.175,A -85,B 0,C 180,E1 -22338.821,E2 -22338.821} C_VEL
LIN {X 0,Y 185.54,Z 292.182,A -85,B 0,C 180,E1 -22344.624,E2 -22344.624} C_VEL
LIN {X 0,Y 185.539,Z 292.189,A -85,B 0,C 180,E1 -22349.5,E2 -22349.5} C_VEL
LIN {X 0,Y 185.492,Z 292.195,A -85,B 0,C 180,E1 -22354.633,E2 -22354.633} C_VEL
LIN {X 0,Y 185.495,Z 292.195,A -85,B 0,C 180,E1 -22357.315,E2 -22357.315} C_VEL
LIN {X 0,Y 185.457,Z 292.2,A -85,B 0,C 180,E1 -22360.722,E2 -22360.722} C_VEL
LIN {X 0,Y 185.452,Z 292.2,A -85,B 0,C 180,E1 -22366.057,E2 -22366.057} C_VEL
LIN {X 0,Y 185.47,Z 292.36,A -85,B 0,C 180,E1 -22369.465,E2 -22369.465} C_VEL
LIN {X 0,Y 186.98,Z 298.162,A -85,B 0,C 180,E1 -22373.032,E2 -22373.032} C_VEL
LIN {X 0,Y 187.657,Z 301.135,A -85,B 0,C 180,E1 -22374.756,E2 -22374.756} C_VEL
LIN {X 0,Y 194.834,Z 317.299,A -85,B 0,C 180,E1 -22376.911,E2 -22376.911} C_VEL
LIN {X 0,Y 197.571,Z 324.756,A -85,B 0,C 180,E1 -22377.733,E2 -22377.733} C_VEL
LIN {X 0,Y 200.359,Z 346.711,A -85,B 0,C 180,E1 -22379.127,E2 -22379.127} C_VEL
LIN {X 0,Y 201.516,Z 358.73,A -85,B 0,C 180,E1 -22379.805,E2 -22379.805} C_VEL
LIN {X 0,Y 200.574,Z 380.863,A -85,B 0,C 180,E1 -22380.625,E2 -22380.625} C_VEL
LIN {X 0,Y 199.662,Z 390.687,A -85,B 0,C 180,E1 -22381.234,E2 -22381.234} C_VEL
LIN {X 0,Y 198.623,Z 394.487,A -85,B 0,C 180,E1 -22381.431,E2 -22381.431} C_VEL
LIN {X 0,Y 195.235,Z 400.325,A -85,B 0,C 180,E1 -22381.595,E2 -22381.595} C_VEL
LIN {X 0,Y 191.625,Z 405.957,A -85,B 0,C 180,E1 -22381.899,E2 -22381.899} C_VEL
LIN {X 0,Y 190.246,Z 409.43,A -85,B 0,C 180,E1 -22382.322,E2 -22382.322} C_VEL
LIN {X 0,Y 187.981,Z 419.007,A -85,B 0,C 180,E1 -22383.963,E2 -22383.963} C_VEL
LIN {X 0,Y 185.917,Z 426.999,A -85,B 0,C 180,E1 -22385.728,E2 -22385.728} C_VEL
LIN {X 0,Y 183.946,Z 433.671,A -85,B 0,C 180,E1 -22387.54,E2 -22387.54} C_VEL
LIN {X 0,Y 182.084,Z 440.02,A -85,B 0,C 180,E1 -22389.674,E2 -22389.674} C_VEL
LIN {X 0,Y 180.398,Z 445.296,A -85,B 0,C 180,E1 -22391.842,E2 -22391.842} C_VEL
LIN {X 0,Y 178.959,Z 449.699,A -85,B 0,C 180,E1 -22394.045,E2 -22394.045} C_VEL
LIN {X 0,Y 177.464,Z 454.912,A -85,B 0,C 180,E1 -22397.421,E2 -22397.421} C_VEL
LIN {X 0,Y 176.572,Z 458.752,A -85,B 0,C 180,E1 -22400.84,E2 -22400.84} C_VEL
LIN {X 0,Y 176.242,Z 460.52,A -85,B 0,C 180,E1 -22403.13,E2 -22403.13} C_VEL
LIN {X 0,Y 176.162,Z 461.976,A -85,B 0,C 180,E1 -22405.846,E2 -22405.846} C_VEL
LIN {X 0,Y 176.249,Z 462.589,A -85,B 0,C 180,E1 -22407.716,E2 -22407.716} C_VEL
LIN {X 0,Y 176.45,Z 462.898,A -85,B 0,C 180,E1 -22410.001,E2 -22410.001} C_VEL
LIN {X 0,Y 176.252,Z 462.579,A -85,B 0,C 180,E1 -22412.286,E2 -22412.286} C_VEL
LIN {X 0,Y 176.148,Z 461.762,A -85,B 0,C 180,E1 -22414.578,E2 -22414.578} C_VEL
LIN {X 0,Y 176.243,Z 460.469,A -85,B 0,C 180,E1 -22416.872,E2 -22416.872} C_VEL
LIN {X 0,Y 176.82,Z 457.509,A -85,B 0,C 180,E1 -22420.304,E2 -22420.304} C_VEL
LIN {X 0,Y 177.465,Z 454.817,A -85,B 0,C 180,E1 -22422.582,E2 -22422.582} C_VEL
LIN {X 0,Y 178.959,Z 449.577,A -85,B 0,C 180,E1 -22425.957,E2 -22425.957} C_VEL
LIN {X 0,Y 181.167,Z 442.686,A -85,B 0,C 180,E1 -22429.254,E2 -22429.254} C_VEL
LIN {X 0,Y 183.418,Z 435.17,A -85,B 0,C 180,E1 -22431.938,E2 -22431.938} C_VEL
LIN {X 0,Y 185.669,Z 427.774,A -85,B 0,C 180,E1 -22434.012,E2 -22434.012} C_VEL
LIN {X 0,Y 187.712,Z 419.942,A -85,B 0,C 180,E1 -22435.779,E2 -22435.779} C_VEL
LIN {X 0,Y 189.603,Z 411.626,A -85,B 0,C 180,E1 -22437.274,E2 -22437.274} C_VEL
LIN {X 0,Y 191.755,Z 400.757,A -85,B 0,C 180,E1 -22438.755,E2 -22438.755} C_VEL
LIN {X 0,Y 193.433,Z 389.882,A -85,B 0,C 180,E1 -22439.748,E2 -22439.748} C_VEL
LIN {X 0,Y 194.343,Z 380.455,A -85,B 0,C 180,E1 -22440.342,E2 -22440.342} C_VEL
LIN {X 0,Y 195.185,Z 358.781,A -85,B 0,C 180,E1 -22441.189,E2 -22441.189} C_VEL
LIN {X 0,Y 192.383,Z 332.071,A -85,B 0,C 180,E1 -22442.837,E2 -22442.837} C_VEL
LIN {X 0,Y 191.236,Z 325.592,A -85,B 0,C 180,E1 -22443.339,E2 -22443.339} C_VEL
LIN {X 0,Y 186.007,Z 312.832,A -85,B 0,C 180,E1 -22444.973,E2 -22444.973} C_VEL
LIN {X 0,Y 181.982,Z 304.349,A -85,B 0,C 180,E1 -22446.254,E2 -22446.254} C_VEL
LIN {X 0,Y 180.327,Z 300.572,A -85,B 0,C 180,E1 -22446.848,E2 -22446.848} C_VEL
LIN {X 0,Y 178.402,Z 293.077,A -85,B 0,C 180,E1 -22451.695,E2 -22451.695} C_VEL
LIN {X 0,Y 178.392,Z 293.08,A -85,B 0,C 180,E1 -22455.166,E2 -22455.166} C_VEL
LIN {X 0,Y 178.398,Z 293.079,A -85,B 0,C 180,E1 -22458.463,E2 -22458.463} C_VEL
LIN {X 0,Y 178.42,Z 293.075,A -85,B 0,C 180,E1 -22463.783,E2 -22463.783} C_VEL
LIN {X 0,Y 178.485,Z 293.068,A -85,B 0,C 180,E1 -22466.547,E2 -22466.547} C_VEL
LIN {X 0,Y 178.425,Z 293.07,A -85,B 0,C 180,E1 -22471.793,E2 -22471.793} C_VEL
LIN {X 0,Y 178.465,Z 293.067,A -85,B 0,C 180,E1 -22476.809,E2 -22476.809} C_VEL
LIN {X 0,Y 178.607,Z 293.049,A -85,B 0,C 180,E1 -22481.652,E2 -22481.652} C_VEL
LIN {X 0,Y 178.626,Z 293.047,A -85,B 0,C 180,E1 -22486.346,E2 -22486.346} C_VEL
LIN {X 0,Y 178.904,Z 292.982,A -85,B 0,C 180,E1 -22490.96,E2 -22490.96} C_VEL
LIN {X 0,Y 179.123,Z 292.986,A -85,B 0,C 180,E1 -22497.752,E2 -22497.752} C_VEL
LIN {X 0,Y 179.347,Z 292.95,A -85,B 0,C 180,E1 -22500,E2 -22500} C_VEL
LIN {X 0,Y 178.83,Z 292.99,A -85,B 0,C 180,E1 -22504.508,E2 -22504.508} C_VEL
LIN {X 0,Y 178.906,Z 293.012,A -85,B 0,C 180,E1 -22509.041,E2 -22509.041} C_VEL
LIN {X 0,Y 178.627,Z 293.022,A -85,B 0,C 180,E1 -22513.655,E2 -22513.655} C_VEL
LIN {X 0,Y 178.557,Z 293.053,A -85,B 0,C 180,E1 -22519.152,E2 -22519.152} C_VEL
LIN {X 0,Y 178.468,Z 293.067,A -85,B 0,C 180,E1 -22525.076,E2 -22525.076} C_VEL
LIN {X 0,Y 178.463,Z 293.067,A -85,B 0,C 180,E1 -22530.794,E2 -22530.794} C_VEL
LIN {X 0,Y 178.485,Z 293.042,A -85,B 0,C 180,E1 -22534.217,E2 -22534.217} C_VEL
LIN {X 0,Y 178.389,Z 293.078,A -85,B 0,C 180,E1 -22539.077,E2 -22539.077} C_VEL
LIN {X 0,Y 178.394,Z 293.061,A -85,B 0,C 180,E1 -22542.047,E2 -22542.047} C_VEL
LIN {X 0,Y 178.393,Z 293.078,A -85,B 0,C 180,E1 -22545.164,E2 -22545.164} C_VEL
LIN {X 0,Y 178.399,Z 293.059,A -85,B 0,C 180,E1 -22548.461,E2 -22548.461} C_VEL
LIN {X 0,Y 178.466,Z 293.023,A -85,B 0,C 180,E1 -22553.17,E2 -22553.17} C_VEL
LIN {X 0,Y 179.455,Z 295.874,A -85,B 0,C 180,E1 -22553.569,E2 -22553.569} C_VEL
LIN {X 0,Y 181.068,Z 298.188,A -85,B 0,C 180,E1 -22554.062,E2 -22554.062} C_VEL
LIN {X 0,Y 188.489,Z 311.055,A -85,B 0,C 180,E1 -22556.287,E2 -22556.287} C_VEL
LIN {X 0,Y 195.803,Z 325.941,A -85,B 0,C 180,E1 -22558.359,E2 -22558.359} C_VEL
LIN {X 0,Y 196.628,Z 327.843,A -85,B 0,C 180,E1 -22558.589,E2 -22558.589} C_VEL
LIN {X 0,Y 195.205,Z 359.807,A -85,B 0,C 180,E1 -22559.731,E2 -22559.731} C_VEL
LIN {X 0,Y 194.564,Z 369.007,A -85,B 0,C 180,E1 -22560.283,E2 -22560.283} C_VEL
LIN {X 0,Y 193.771,Z 377.494,A -85,B 0,C 180,E1 -22561.043,E2 -22561.043} C_VEL
LIN {X 0,Y 192.679,Z 385.609,A -85,B 0,C 180,E1 -22561.989,E2 -22561.989} C_VEL
LIN {X 0,Y 191.075,Z 394.022,A -85,B 0,C 180,E1 -22563.219,E2 -22563.219} C_VEL
LIN {X 0,Y 189.286,Z 402.109,A -85,B 0,C 180,E1 -22564.723,E2 -22564.723} C_VEL
LIN {X 0,Y 187.392,Z 409.786,A -85,B 0,C 180,E1 -22566.516,E2 -22566.516} C_VEL
LIN {X 0,Y 185.193,Z 417.81,A -85,B 0,C 180,E1 -22568.867,E2 -22568.867} C_VEL
LIN {X 0,Y 182.971,Z 424.835,A -85,B 0,C 180,E1 -22571.524,E2 -22571.524} C_VEL
LIN {X 0,Y 181.041,Z 430.383,A -85,B 0,C 180,E1 -22574.231,E2 -22574.231} C_VEL
LIN {X 0,Y 179.309,Z 435.528,A -85,B 0,C 180,E1 -22577.55,E2 -22577.55} C_VEL
LIN {X 0,Y 178.193,Z 438.792,A -85,B 0,C 180,E1 -22580.407,E2 -22580.407} C_VEL
LIN {X 0,Y 177.393,Z 441.052,A -85,B 0,C 180,E1 -22583.173,E2 -22583.173} C_VEL
LIN {X 0,Y 176.937,Z 442.311,A -85,B 0,C 180,E1 -22585.442,E2 -22585.442} C_VEL
LIN {X 0,Y 176.634,Z 443.105,A -85,B 0,C 180,E1 -22587.719,E2 -22587.719} C_VEL
LIN {X 0,Y 176.528,Z 443.408,A -85,B 0,C 180,E1 -22589.999,E2 -22589.999} C_VEL
LIN {X 0,Y 176.631,Z 443.128,A -85,B 0,C 180,E1 -22592.279,E2 -22592.279} C_VEL
LIN {X 0,Y 176.908,Z 442.38,A -85,B 0,C 180,E1 -22594.556,E2 -22594.556} C_VEL
LIN {X 0,Y 177.383,Z 441.167,A -85,B 0,C 180,E1 -22596.825,E2 -22596.825} C_VEL
LIN {X 0,Y 178.191,Z 438.954,A -85,B 0,C 180,E1 -22599.591,E2 -22599.591} C_VEL
LIN {X 0,Y 179.277,Z 435.743,A -85,B 0,C 180,E1 -22602.45,E2 -22602.45} C_VEL
LIN {X 0,Y 181.012,Z 430.655,A -85,B 0,C 180,E1 -22605.769,E2 -22605.769} C_VEL
LIN {X 0,Y 182.912,Z 425.172,A -85,B 0,C 180,E1 -22608.48,E2 -22608.48} C_VEL
LIN {X 0,Y 185.166,Z 418.271,A -85,B 0,C 180,E1 -22611.134,E2 -22611.134} C_VEL
LIN {X 0,Y 187.323,Z 410.353,A -85,B 0,C 180,E1 -22613.491,E2 -22613.491} C_VEL
LIN {X 0,Y 189.238,Z 402.794,A -85,B 0,C 180,E1 -22615.282,E2 -22615.282} C_VEL
LIN {X 0,Y 191.073,Z 394.859,A -85,B 0,C 180,E1 -22616.779,E2 -22616.779} C_VEL
LIN {X 0,Y 192.603,Z 386.656,A -85,B 0,C 180,E1 -22618.02,E2 -22618.02} C_VEL
LIN {X 0,Y 193.764,Z 378.884,A -85,B 0,C 180,E1 -22618.951,E2 -22618.951} C_VEL
LIN {X 0,Y 194.684,Z 369.685,A -85,B 0,C 180,E1 -22619.799,E2 -22619.799} C_VEL
LIN {X 0,Y 195.323,Z 360.112,A -85,B 0,C 180,E1 -22620.396,E2 -22620.396} C_VEL
LIN {X 0,Y 196.676,Z 327.898,A -85,B 0,C 180,E1 -22621.565,E2 -22621.565} C_VEL
LIN {X 0,Y 190.245,Z 314.336,A -85,B 0,C 180,E1 -22623.381,E2 -22623.381} C_VEL
LIN {X 0,Y 183.923,Z 303.052,A -85,B 0,C 180,E1 -22625.236,E2 -22625.236} C_VEL
LIN {X 0,Y 180.245,Z 296.927,A -85,B 0,C 180,E1 -22626.376,E2 -22626.376} C_VEL
LIN {X 0,Y 178.784,Z 294.443,A -85,B 0,C 180,E1 -22626.849,E2 -22626.849} C_VEL
LIN {X 0,Y 178.455,Z 293.06,A -85,B 0,C 180,E1 -22627.017,E2 -22627.017} C_VEL
LIN {X 0,Y 178.39,Z 293.062,A -85,B 0,C 180,E1 -22632.046,E2 -22632.046} C_VEL
LIN {X 0,Y 178.388,Z 293.075,A -85,B 0,C 180,E1 -22635.164,E2 -22635.164} C_VEL
LIN {X 0,Y 178.393,Z 293.056,A -85,B 0,C 180,E1 -22638.461,E2 -22638.461} C_VEL
LIN {X 0,Y 178.415,Z 293.066,A -85,B 0,C 180,E1 -22643.781,E2 -22643.781} C_VEL
LIN {X 0,Y 178.48,Z 293.061,A -85,B 0,C 180,E1 -22646.545,E2 -22646.545} C_VEL
LIN {X 0,Y 178.439,Z 293.063,A -85,B 0,C 180,E1 -22651.794,E2 -22651.794} C_VEL
LIN {X 0,Y 178.512,Z 293.061,A -85,B 0,C 180,E1 -22654.888,E2 -22654.888} C_VEL
LIN {X 0,Y 178.601,Z 293.045,A -85,B 0,C 180,E1 -22661.651,E2 -22661.651} C_VEL
LIN {X 0,Y 178.621,Z 293.022,A -85,B 0,C 180,E1 -22666.345,E2 -22666.345} C_VEL
LIN {X 0,Y 178.899,Z 293.013,A -85,B 0,C 180,E1 -22670.959,E2 -22670.959} C_VEL
LIN {X 0,Y 179.117,Z 292.96,A -85,B 0,C 180,E1 -22677.751,E2 -22677.751} C_VEL
LIN {X 0,Y 179.34,Z 292.952,A -85,B 0,C 180,E1 -22680,E2 -22680} C_VEL
LIN {X 0,Y 178.827,Z 293.015,A -85,B 0,C 180,E1 -22684.508,E2 -22684.508} C_VEL
LIN {X 0,Y 178.901,Z 293.01,A -85,B 0,C 180,E1 -22689.041,E2 -22689.041} C_VEL
LIN {X 0,Y 178.621,Z 293.048,A -85,B 0,C 180,E1 -22693.655,E2 -22693.655} C_VEL
LIN {X 0,Y 178.55,Z 293.055,A -85,B 0,C 180,E1 -22699.152,E2 -22699.152} C_VEL
LIN {X 0,Y 178.461,Z 293.064,A -85,B 0,C 180,E1 -22705.077,E2 -22705.077} C_VEL
LIN {X 0,Y 178.456,Z 293.071,A -85,B 0,C 180,E1 -22710.795,E2 -22710.795} C_VEL
LIN {X 0,Y 178.478,Z 293.069,A -85,B 0,C 180,E1 -22714.218,E2 -22714.218} C_VEL
LIN {X 0,Y 178.383,Z 293.081,A -85,B 0,C 180,E1 -22719.077,E2 -22719.077} C_VEL
LIN {X 0,Y 178.389,Z 293.08,A -85,B 0,C 180,E1 -22722.047,E2 -22722.047} C_VEL
LIN {X 0,Y 178.387,Z 293.08,A -85,B 0,C 180,E1 -22725.166,E2 -22725.166} C_VEL
LIN {X 0,Y 178.397,Z 293.182,A -85,B 0,C 180,E1 -22728.307,E2 -22728.307} C_VEL
LIN {X 0,Y 180.325,Z 300.654,A -85,B 0,C 180,E1 -22733.093,E2 -22733.093} C_VEL
LIN {X 0,Y 182.263,Z 304.816,A -85,B 0,C 180,E1 -22733.742,E2 -22733.742} C_VEL
LIN {X 0,Y 188.098,Z 317.526,A -85,B 0,C 180,E1 -22735.593,E2 -22735.593} C_VEL
LIN {X 0,Y 191.695,Z 326.758,A -85,B 0,C 180,E1 -22736.721,E2 -22736.721} C_VEL
LIN {X 0,Y 194.29,Z 347.988,A -85,B 0,C 180,E1 -22738.121,E2 -22738.121} C_VEL
LIN {X 0,Y 195.348,Z 360.208,A -85,B 0,C 180,E1 -22738.825,E2 -22738.825} C_VEL
LIN {X 0,Y 194.406,Z 380.486,A -85,B 0,C 180,E1 -22739.596,E2 -22739.596} C_VEL
LIN {X 0,Y 193.321,Z 391.551,A -85,B 0,C 180,E1 -22740.31,E2 -22740.31} C_VEL
LIN {X 0,Y 191.417,Z 403.175,A -85,B 0,C 180,E1 -22741.492,E2 -22741.492} C_VEL
LIN {X 0,Y 190.246,Z 409.43,A -85,B 0,C 180,E1 -22742.322,E2 -22742.322} C_VEL
LIN {X 0,Y 188.452,Z 414.712,A -85,B 0,C 180,E1 -22743.082,E2 -22743.082} C_VEL
LIN {X 0,Y 183.821,Z 422.613,A -85,B 0,C 180,E1 -22744.268,E2 -22744.268} C_VEL
LIN {X 0,Y 179.099,Z 429.907,A -85,B 0,C 180,E1 -22745.725,E2 -22745.725} C_VEL
LIN {X 0,Y 177.168,Z 433.998,A -85,B 0,C 180,E1 -22746.889,E2 -22746.889} C_VEL
LIN {X 0,Y 174.953,Z 441.057,A -85,B 0,C 180,E1 -22749.423,E2 -22749.423} C_VEL
LIN {X 0,Y 172.502,Z 448.344,A -85,B 0,C 180,E1 -22752.821,E2 -22752.821} C_VEL
LIN {X 0,Y 170.992,Z 452.983,A -85,B 0,C 180,E1 -22755.724,E2 -22755.724} C_VEL
LIN {X 0,Y 170.117,Z 456.005,A -85,B 0,C 180,E1 -22758.08,E2 -22758.08} C_VEL
LIN {X 0,Y 169.541,Z 458.359,A -85,B 0,C 180,E1 -22760.457,E2 -22760.457} C_VEL
LIN {X 0,Y 169.171,Z 460.128,A -85,B 0,C 180,E1 -22762.842,E2 -22762.842} C_VEL
LIN {X 0,Y 169.086,Z 461.714,A -85,B 0,C 180,E1 -22765.984,E2 -22765.984} C_VEL
LIN {X 0,Y 169.361,Z 462.506,A -85,B 0,C 180,E1 -22770.001,E2 -22770.001} C_VEL
LIN {X 0,Y 169.088,Z 461.681,A -85,B 0,C 180,E1 -22774.022,E2 -22774.022} C_VEL
LIN {X 0,Y 169.172,Z 460.075,A -85,B 0,C 180,E1 -22777.161,E2 -22777.161} C_VEL
LIN {X 0,Y 169.799,Z 457.114,A -85,B 0,C 180,E1 -22780.736,E2 -22780.736} C_VEL
LIN {X 0,Y 170.514,Z 454.422,A -85,B 0,C 180,E1 -22783.104,E2 -22783.104} C_VEL
LIN {X 0,Y 172.123,Z 449.182,A -85,B 0,C 180,E1 -22786.609,E2 -22786.609} C_VEL
LIN {X 0,Y 174.469,Z 442.292,A -85,B 0,C 180,E1 -22790.024,E2 -22790.024} C_VEL
LIN {X 0,Y 176.839,Z 434.775,A -85,B 0,C 180,E1 -22792.799,E2 -22792.799} C_VEL
LIN {X 0,Y 179.197,Z 427.378,A -85,B 0,C 180,E1 -22794.937,E2 -22794.937} C_VEL
LIN {X 0,Y 181.094,Z 420.517,A -85,B 0,C 180,E1 -22796.55,E2 -22796.55} C_VEL
LIN {X 0,Y 183.01,Z 412.579,A -85,B 0,C 180,E1 -22798.063,E2 -22798.063} C_VEL
LIN {X 0,Y 184.828,Z 404.177,A -85,B 0,C 180,E1 -22799.313,E2 -22799.313} C_VEL
LIN {X 0,Y 186.375,Z 395.585,A -85,B 0,C 180,E1 -22800.29,E2 -22800.29} C_VEL
LIN {X 0,Y 187.806,Z 385.318,A -85,B 0,C 180,E1 -22801.125,E2 -22801.125} C_VEL
LIN {X 0,Y 188.763,Z 370.657,A -85,B 0,C 180,E1 -22801.837,E2 -22801.837} C_VEL
LIN {X 0,Y 189.114,Z 359.733,A -85,B 0,C 180,E1 -22802.249,E2 -22802.249} C_VEL
LIN {X 0,Y 186.525,Z 333.868,A -85,B 0,C 180,E1 -22803.906,E2 -22803.906} C_VEL
LIN {X 0,Y 185.546,Z 328.237,A -85,B 0,C 180,E1 -22804.364,E2 -22804.364} C_VEL
LIN {X 0,Y 180.62,Z 316.14,A -85,B 0,C 180,E1 -22806,E2 -22806} C_VEL
LIN {X 0,Y 176.52,Z 307.485,A -85,B 0,C 180,E1 -22807.388,E2 -22807.388} C_VEL
LIN {X 0,Y 174.536,Z 303.62,A -85,B 0,C 180,E1 -22808.077,E2 -22808.077} C_VEL
LIN {X 0,Y 172.902,Z 300.049,A -85,B 0,C 180,E1 -22808.72,E2 -22808.72} C_VEL
LIN {X 0,Y 171.324,Z 293.96,A -85,B 0,C 180,E1 -22812.914,E2 -22812.914} C_VEL
LIN {X 0,Y 171.333,Z 293.958,A -85,B 0,C 180,E1 -22817.593,E2 -22817.593} C_VEL
LIN {X 0,Y 171.361,Z 293.955,A -85,B 0,C 180,E1 -22822.034,E2 -22822.034} C_VEL
LIN {X 0,Y 171.399,Z 293.949,A -85,B 0,C 180,E1 -22825.094,E2 -22825.094} C_VEL
LIN {X 0,Y 171.394,Z 293.949,A -85,B 0,C 180,E1 -22830.524,E2 -22830.524} C_VEL
LIN {X 0,Y 171.405,Z 293.944,A -85,B 0,C 180,E1 -22835.794,E2 -22835.794} C_VEL
LIN {X 0,Y 171.511,Z 293.932,A -85,B 0,C 180,E1 -22840.864,E2 -22840.864} C_VEL
LIN {X 0,Y 171.542,Z 293.929,A -85,B 0,C 180,E1 -22845.77,E2 -22845.77} C_VEL
LIN {X 0,Y 171.843,Z 293.863,A -85,B 0,C 180,E1 -22850.585,E2 -22850.585} C_VEL
LIN {X 0,Y 171.779,Z 293.889,A -85,B 0,C 180,E1 -22855.307,E2 -22855.307} C_VEL
LIN {X 0,Y 172.311,Z 293.826,A -85,B 0,C 180,E1 -22860,E2 -22860} C_VEL
LIN {X 0,Y 171.841,Z 293.879,A -85,B 0,C 180,E1 -22866.85,E2 -22866.85} C_VEL
LIN {X 0,Y 171.769,Z 293.898,A -85,B 0,C 180,E1 -22870.892,E2 -22870.892} C_VEL
LIN {X 0,Y 171.501,Z 293.91,A -85,B 0,C 180,E1 -22876.67,E2 -22876.67} C_VEL
LIN {X 0,Y 171.481,Z 293.937,A -85,B 0,C 180,E1 -22879.498,E2 -22879.498} C_VEL
LIN {X 0,Y 171.406,Z 293.946,A -85,B 0,C 180,E1 -22885.569,E2 -22885.569} C_VEL
LIN {X 0,Y 171.42,Z 293.945,A -85,B 0,C 180,E1 -22890.572,E2 -22890.572} C_VEL
LIN {X 0,Y 171.395,Z 293.923,A -85,B 0,C 180,E1 -22895.035,E2 -22895.035} C_VEL
LIN {X 0,Y 171.345,Z 293.956,A -85,B 0,C 180,E1 -22898.8,E2 -22898.8} C_VEL
LIN {X 0,Y 171.32,Z 293.949,A -85,B 0,C 180,E1 -22904.218,E2 -22904.218} C_VEL
LIN {X 0,Y 171.332,Z 293.928,A -85,B 0,C 180,E1 -22908.979,E2 -22908.979} C_VEL
LIN {X 0,Y 171.388,Z 294.018,A -85,B 0,C 180,E1 -22911.423,E2 -22911.423} C_VEL
LIN {X 0,Y 172.338,Z 296.716,A -85,B 0,C 180,E1 -22911.819,E2 -22911.819} C_VEL
LIN {X 0,Y 174.188,Z 299.224,A -85,B 0,C 180,E1 -22912.432,E2 -22912.432} C_VEL
LIN {X 0,Y 182.025,Z 312.439,A -85,B 0,C 180,E1 -22914.963,E2 -22914.963} C_VEL
LIN {X 0,Y 189.313,Z 327.042,A -85,B 0,C 180,E1 -22917.17,E2 -22917.17} C_VEL
LIN {X 0,Y 190.49,Z 329.713,A -85,B 0,C 180,E1 -22917.519,E2 -22917.519} C_VEL
LIN {X 0,Y 189.131,Z 360.214,A -85,B 0,C 180,E1 -22918.651,E2 -22918.651} C_VEL
LIN {X 0,Y 188.421,Z 369.709,A -85,B 0,C 180,E1 -22919.24,E2 -22919.24} C_VEL
LIN {X 0,Y 187.569,Z 378.338,A -85,B 0,C 180,E1 -22920.046,E2 -22920.046} C_VEL
LIN {X 0,Y 186.465,Z 386.005,A -85,B 0,C 180,E1 -22920.969,E2 -22920.969} C_VEL
LIN {X 0,Y 184.796,Z 394.417,A -85,B 0,C 180,E1 -22922.232,E2 -22922.232} C_VEL
LIN {X 0,Y 182.912,Z 402.504,A -85,B 0,C 180,E1 -22923.776,E2 -22923.776} C_VEL
LIN {X 0,Y 180.93,Z 410.179,A -85,B 0,C 180,E1 -22925.623,E2 -22925.623} C_VEL
LIN {X 0,Y 178.62,Z 418.203,A -85,B 0,C 180,E1 -22928.049,E2 -22928.049} C_VEL
LIN {X 0,Y 176.279,Z 425.227,A -85,B 0,C 180,E1 -22930.796,E2 -22930.796} C_VEL
LIN {X 0,Y 174.246,Z 430.775,A -85,B 0,C 180,E1 -22933.599,E2 -22933.599} C_VEL
LIN {X 0,Y 172.391,Z 435.921,A -85,B 0,C 180,E1 -22937.042,E2 -22937.042} C_VEL
LIN {X 0,Y 171.118,Z 439.465,A -85,B 0,C 180,E1 -22940.302,E2 -22940.302} C_VEL
LIN {X 0,Y 170.369,Z 441.443,A -85,B 0,C 180,E1 -22942.89,E2 -22942.89} C_VEL
LIN {X 0,Y 169.879,Z 442.702,A -85,B 0,C 180,E1 -22945.253,E2 -22945.253} C_VEL
LIN {X 0,Y 169.557,Z 443.496,A -85,B 0,C 180,E1 -22947.623,E2 -22947.623} C_VEL
LIN {X 0,Y 169.468,Z 443.798,A -85,B 0,C 180,E1 -22949.999,E2 -22949.999} C_VEL
LIN {X 0,Y 169.553,Z 443.519,A -85,B 0,C 180,E1 -22952.374,E2 -22952.374} C_VEL
LIN {X 0,Y 169.852,Z 442.771,A -85,B 0,C 180,E1 -22954.746,E2 -22954.746} C_VEL
LIN {X 0,Y 170.359,Z 441.557,A -85,B 0,C 180,E1 -22957.108,E2 -22957.108} C_VEL
LIN {X 0,Y 171.39,Z 438.831,A -85,B 0,C 180,E1 -22960.513,E2 -22960.513} C_VEL
LIN {X 0,Y 172.371,Z 436.132,A -85,B 0,C 180,E1 -22962.957,E2 -22962.957} C_VEL
LIN {X 0,Y 174.214,Z 431.044,A -85,B 0,C 180,E1 -22966.401,E2 -22966.401} C_VEL
LIN {X 0,Y 176.219,Z 425.56,A -85,B 0,C 180,E1 -22969.208,E2 -22969.208} C_VEL
LIN {X 0,Y 178.592,Z 418.659,A -85,B 0,C 180,E1 -22971.952,E2 -22971.952} C_VEL
LIN {X 0,Y 180.851,Z 410.74,A -85,B 0,C 180,E1 -22974.385,E2 -22974.385} C_VEL
LIN {X 0,Y 182.862,Z 403.181,A -85,B 0,C 180,E1 -22976.229,E2 -22976.229} C_VEL
LIN {X 0,Y 184.794,Z 395.244,A -85,B 0,C 180,E1 -22977.766,E2 -22977.766} C_VEL
LIN {X 0,Y 186.388,Z 387.041,A -85,B 0,C 180,E1 -22979.042,E2 -22979.042} C_VEL
LIN {X 0,Y 187.778,Z 378.065,A -85,B 0,C 180,E1 -22980.12,E2 -22980.12} C_VEL
LIN {X 0,Y 188.688,Z 368.478,A -85,B 0,C 180,E1 -22980.997,E2 -22980.997} C_VEL
LIN {X 0,Y 189.441,Z 357.356,A -85,B 0,C 180,E1 -22981.633,E2 -22981.633} C_VEL
LIN {X 0,Y 190.654,Z 330.054,A -85,B 0,C 180,E1 -22982.605,E2 -22982.605} C_VEL
LIN {X 0,Y 183.439,Z 315.002,A -85,B 0,C 180,E1 -22984.782,E2 -22984.782} C_VEL
LIN {X 0,Y 175.735,Z 301.771,A -85,B 0,C 180,E1 -22987.236,E2 -22987.236} C_VEL
LIN {X 0,Y 173.372,Z 298.057,A -85,B 0,C 180,E1 -22988.032,E2 -22988.032} C_VEL
LIN {X 0,Y 171.781,Z 295.661,A -85,B 0,C 180,E1 -22988.58,E2 -22988.58} C_VEL
LIN {X 0,Y 171.35,Z 293.954,A -85,B 0,C 180,E1 -22988.804,E2 -22988.804} C_VEL
LIN {X 0,Y 171.315,Z 293.957,A -85,B 0,C 180,E1 -22994.217,E2 -22994.217} C_VEL
LIN {X 0,Y 171.326,Z 293.938,A -85,B 0,C 180,E1 -22998.978,E2 -22998.978} C_VEL
LIN {X 0,Y 171.356,Z 293.949,A -85,B 0,C 180,E1 -23002.032,E2 -23002.032} C_VEL
LIN {X 0,Y 171.394,Z 293.944,A -85,B 0,C 180,E1 -23005.092,E2 -23005.092} C_VEL
LIN {X 0,Y 171.405,Z 293.944,A -85,B 0,C 180,E1 -23010.526,E2 -23010.526} C_VEL
LIN {X 0,Y 171.432,Z 293.941,A -85,B 0,C 180,E1 -23015.798,E2 -23015.798} C_VEL
LIN {X 0,Y 171.503,Z 293.933,A -85,B 0,C 180,E1 -23020.863,E2 -23020.863} C_VEL
LIN {X 0,Y 171.537,Z 293.899,A -85,B 0,C 180,E1 -23025.769,E2 -23025.769} C_VEL
LIN {X 0,Y 171.838,Z 293.893,A -85,B 0,C 180,E1 -23030.584,E2 -23030.584} C_VEL
LIN {X 0,Y 171.774,Z 293.869,A -85,B 0,C 180,E1 -23035.306,E2 -23035.306} C_VEL
LIN {X 0,Y 172.305,Z 293.828,A -85,B 0,C 180,E1 -23040,E2 -23040} C_VEL
LIN {X 0,Y 171.777,Z 293.892,A -85,B 0,C 180,E1 -23044.693,E2 -23044.693} C_VEL
LIN {X 0,Y 171.839,Z 293.889,A -85,B 0,C 180,E1 -23049.415,E2 -23049.415} C_VEL
LIN {X 0,Y 171.537,Z 293.929,A -85,B 0,C 180,E1 -23054.23,E2 -23054.23} C_VEL
LIN {X 0,Y 171.475,Z 293.936,A -85,B 0,C 180,E1 -23059.5,E2 -23059.5} C_VEL
LIN {X 0,Y 171.399,Z 293.946,A -85,B 0,C 180,E1 -23065.57,E2 -23065.57} C_VEL
LIN {X 0,Y 171.413,Z 293.948,A -85,B 0,C 180,E1 -23070.573,E2 -23070.573} C_VEL
LIN {X 0,Y 171.388,Z 293.953,A -85,B 0,C 180,E1 -23075.036,E2 -23075.036} C_VEL
LIN {X 0,Y 171.339,Z 293.959,A -85,B 0,C 180,E1 -23078.802,E2 -23078.802} C_VEL
LIN {X 0,Y 171.314,Z 293.961,A -85,B 0,C 180,E1 -23084.219,E2 -23084.219} C_VEL
LIN {X 0,Y 171.326,Z 294.085,A -85,B 0,C 180,E1 -23087.085,E2 -23087.085} C_VEL
LIN {X 0,Y 172.996,Z 300.337,A -85,B 0,C 180,E1 -23091.256,E2 -23091.256} C_VEL
LIN {X 0,Y 175.216,Z 304.659,A -85,B 0,C 180,E1 -23092.048,E2 -23092.048} C_VEL
LIN {X 0,Y 181.481,Z 317.962,A -85,B 0,C 180,E1 -23094.191,E2 -23094.191} C_VEL
LIN {X 0,Y 186.023,Z 329.674,A -85,B 0,C 180,E1 -23095.716,E2 -23095.716} C_VEL
LIN {X 0,Y 188.821,Z 354.515,A -85,B 0,C 180,E1 -23097.386,E2 -23097.386} C_VEL
LIN {X 0,Y 189.214,Z 362.471,A -85,B 0,C 180,E1 -23097.81,E2 -23097.81} C_VEL
LIN {X 0,Y 188.224,Z 381.408,A -85,B 0,C 180,E1 -23098.564,E2 -23098.564} C_VEL
LIN {X 0,Y 186.799,Z 393.796,A -85,B 0,C 180,E1 -23099.476,E2 -23099.476} C_VEL
LIN {X 0,Y 185.207,Z 402.788,A -85,B 0,C 180,E1 -23100.443,E2 -23100.443} C_VEL
LIN {X 0,Y 183.391,Z 411.474,A -85,B 0,C 180,E1 -23101.693,E2 -23101.693} C_VEL
LIN {X 0,Y 181.277,Z 419.997,A -85,B 0,C 180,E1 -23103.271,E2 -23103.271} C_VEL
LIN {X 0,Y 179.177,Z 427.635,A -85,B 0,C 180,E1 -23105.062,E2 -23105.062} C_VEL
LIN {X 0,Y 177.168,Z 433.998,A -85,B 0,C 180,E1 -23106.889,E2 -23106.889} C_VEL
LIN {X 0,Y 175.234,Z 438.031,A -85,B 0,C 180,E1 -23108.17,E2 -23108.17} C_VEL
LIN {X 0,Y 170.48,Z 443.878,A -85,B 0,C 180,E1 -23110.308,E2 -23110.308} C_VEL
LIN {X 0,Y 165.936,Z 448.997,A -85,B 0,C 180,E1 -23112.756,E2 -23112.756} C_VEL
LIN {X 0,Y 164.374,Z 451.696,A -85,B 0,C 180,E1 -23114.485,E2 -23114.485} C_VEL
LIN {X 0,Y 163.162,Z 455.613,A -85,B 0,C 180,E1 -23117.564,E2 -23117.564} C_VEL
LIN {X 0,Y 162.528,Z 457.967,A -85,B 0,C 180,E1 -23120.041,E2 -23120.041} C_VEL
LIN {X 0,Y 162.126,Z 459.736,A -85,B 0,C 180,E1 -23122.529,E2 -23122.529} C_VEL
LIN {X 0,Y 161.995,Z 461.486,A -85,B 0,C 180,E1 -23126.223,E2 -23126.223} C_VEL
LIN {X 0,Y 162.274,Z 462.115,A -85,B 0,C 180,E1 -23130.001,E2 -23130.001} C_VEL
LIN {X 0,Y 161.999,Z 461.448,A -85,B 0,C 180,E1 -23133.797,E2 -23133.797} C_VEL
LIN {X 0,Y 162.127,Z 459.682,A -85,B 0,C 180,E1 -23137.474,E2 -23137.474} C_VEL
LIN {X 0,Y 162.803,Z 456.72,A -85,B 0,C 180,E1 -23141.203,E2 -23141.203} C_VEL
LIN {X 0,Y 163.586,Z 454.028,A -85,B 0,C 180,E1 -23143.669,E2 -23143.669} C_VEL
LIN {X 0,Y 165.312,Z 448.788,A -85,B 0,C 180,E1 -23147.314,E2 -23147.314} C_VEL
LIN {X 0,Y 167.811,Z 441.897,A -85,B 0,C 180,E1 -23150.855,E2 -23150.855} C_VEL
LIN {X 0,Y 170.31,Z 434.38,A -85,B 0,C 180,E1 -23153.726,E2 -23153.726} C_VEL
LIN {X 0,Y 172.783,Z 426.983,A -85,B 0,C 180,E1 -23155.93,E2 -23155.93} C_VEL
LIN {X 0,Y 174.73,Z 420.198,A -85,B 0,C 180,E1 -23157.578,E2 -23157.578} C_VEL
LIN {X 0,Y 176.758,Z 412.182,A -85,B 0,C 180,E1 -23159.149,E2 -23159.149} C_VEL
LIN {X 0,Y 178.668,Z 403.779,A -85,B 0,C 180,E1 -23160.428,E2 -23160.428} C_VEL
LIN {X 0,Y 180.294,Z 395.187,A -85,B 0,C 180,E1 -23161.425,E2 -23161.425} C_VEL
LIN {X 0,Y 181.662,Z 385.748,A -85,B 0,C 180,E1 -23162.22,E2 -23162.22} C_VEL
LIN {X 0,Y 182.608,Z 373.778,A -85,B 0,C 180,E1 -23162.882,E2 -23162.882} C_VEL
LIN {X 0,Y 183.11,Z 360.315,A -85,B 0,C 180,E1 -23163.397,E2 -23163.397} C_VEL
LIN {X 0,Y 180.522,Z 334.245,A -85,B 0,C 180,E1 -23165.159,E2 -23165.159} C_VEL
LIN {X 0,Y 179.766,Z 330.483,A -85,B 0,C 180,E1 -23165.506,E2 -23165.506} C_VEL
LIN {X 0,Y 174.131,Z 316.721,A -85,B 0,C 180,E1 -23167.513,E2 -23167.513} C_VEL
LIN {X 0,Y 169.742,Z 307.813,A -85,B 0,C 180,E1 -23169.114,E2 -23169.114} C_VEL
LIN {X 0,Y 167.498,Z 303.665,A -85,B 0,C 180,E1 -23169.957,E2 -23169.957} C_VEL
LIN {X 0,Y 165.465,Z 299.48,A -85,B 0,C 180,E1 -23170.838,E2 -23170.838} C_VEL
LIN {X 0,Y 164.27,Z 294.838,A -85,B 0,C 180,E1 -23174.335,E2 -23174.335} C_VEL
LIN {X 0,Y 164.262,Z 294.84,A -85,B 0,C 180,E1 -23176.799,E2 -23176.799} C_VEL
LIN {X 0,Y 164.29,Z 294.836,A -85,B 0,C 180,E1 -23180.356,E2 -23180.356} C_VEL
LIN {X 0,Y 164.327,Z 294.832,A -85,B 0,C 180,E1 -23184.352,E2 -23184.352} C_VEL
LIN {X 0,Y 164.359,Z 294.826,A -85,B 0,C 180,E1 -23189.128,E2 -23189.128} C_VEL
LIN {X 0,Y 164.358,Z 294.824,A -85,B 0,C 180,E1 -23194.685,E2 -23194.685} C_VEL
LIN {X 0,Y 164.419,Z 294.813,A -85,B 0,C 180,E1 -23200.118,E2 -23200.118} C_VEL
LIN {X 0,Y 164.472,Z 294.808,A -85,B 0,C 180,E1 -23205.145,E2 -23205.145} C_VEL
LIN {X 0,Y 164.764,Z 294.747,A -85,B 0,C 180,E1 -23210.176,E2 -23210.176} C_VEL
LIN {X 0,Y 164.818,Z 294.731,A -85,B 0,C 180,E1 -23212.651,E2 -23212.651} C_VEL
LIN {X 0,Y 165.276,Z 294.703,A -85,B 0,C 180,E1 -23220,E2 -23220} C_VEL
LIN {X 0,Y 164.82,Z 294.758,A -85,B 0,C 180,E1 -23227.35,E2 -23227.35} C_VEL
LIN {X 0,Y 164.704,Z 294.776,A -85,B 0,C 180,E1 -23231.057,E2 -23231.057} C_VEL
LIN {X 0,Y 164.426,Z 294.797,A -85,B 0,C 180,E1 -23237.41,E2 -23237.41} C_VEL
LIN {X 0,Y 164.422,Z 294.816,A -85,B 0,C 180,E1 -23239.996,E2 -23239.996} C_VEL
LIN {X 0,Y 164.341,Z 294.826,A -85,B 0,C 180,E1 -23246.094,E2 -23246.094} C_VEL
LIN {X 0,Y 164.36,Z 294.822,A -85,B 0,C 180,E1 -23251.217,E2 -23251.217} C_VEL
LIN {X 0,Y 164.282,Z 294.82,A -85,B 0,C 180,E1 -23256.793,E2 -23256.793} C_VEL
LIN {X 0,Y 164.288,Z 294.833,A -85,B 0,C 180,E1 -23259.917,E2 -23259.917} C_VEL
LIN {X 0,Y 164.282,Z 294.818,A -85,B 0,C 180,E1 -23263.341,E2 -23263.341} C_VEL
LIN {X 0,Y 164.288,Z 294.812,A -85,B 0,C 180,E1 -23268.47,E2 -23268.47} C_VEL
LIN {X 0,Y 164.275,Z 294.809,A -85,B 0,C 180,E1 -23269.43,E2 -23269.43} C_VEL
LIN {X 0,Y 165.193,Z 297.501,A -85,B 0,C 180,E1 -23269.857,E2 -23269.857} C_VEL
LIN {X 0,Y 167.175,Z 300.082,A -85,B 0,C 180,E1 -23270.577,E2 -23270.577} C_VEL
LIN {X 0,Y 174.041,Z 311.299,A -85,B 0,C 180,E1 -23273.011,E2 -23273.011} C_VEL
LIN {X 0,Y 179.977,Z 322.253,A -85,B 0,C 180,E1 -23274.97,E2 -23274.97} C_VEL
LIN {X 0,Y 184.476,Z 331.773,A -85,B 0,C 180,E1 -23276.397,E2 -23276.397} C_VEL
LIN {X 0,Y 183.115,Z 360.623,A -85,B 0,C 180,E1 -23277.497,E2 -23277.497} C_VEL
LIN {X 0,Y 182.364,Z 370.19,A -85,B 0,C 180,E1 -23278.108,E2 -23278.108} C_VEL
LIN {X 0,Y 181.459,Z 378.942,A -85,B 0,C 180,E1 -23278.956,E2 -23278.956} C_VEL
LIN {X 0,Y 179.974,Z 388.268,A -85,B 0,C 180,E1 -23280.139,E2 -23280.139} C_VEL
LIN {X 0,Y 177.853,Z 397.805,A -85,B 0,C 180,E1 -23281.692,E2 -23281.692} C_VEL
LIN {X 0,Y 175.685,Z 406.494,A -85,B 0,C 180,E1 -23283.573,E2 -23283.573} C_VEL
LIN {X 0,Y 173.162,Z 415.213,A -85,B 0,C 180,E1 -23286.054,E2 -23286.054} C_VEL
LIN {X 0,Y 171.054,Z 421.533,A -85,B 0,C 180,E1 -23288.297,E2 -23288.297} C_VEL
LIN {X 0,Y 169.139,Z 426.786,A -85,B 0,C 180,E1 -23290.583,E2 -23290.583} C_VEL
LIN {X 0,Y 167.48,Z 431.167,A -85,B 0,C 180,E1 -23292.917,E2 -23292.917} C_VEL
LIN {X 0,Y 165.507,Z 436.313,A -85,B 0,C 180,E1 -23296.493,E2 -23296.493} C_VEL
LIN {X 0,Y 164.464,Z 438.95,A -85,B 0,C 180,E1 -23298.912,E2 -23298.912} C_VEL
LIN {X 0,Y 163.35,Z 441.835,A -85,B 0,C 180,E1 -23302.583,E2 -23302.583} C_VEL
LIN {X 0,Y 162.824,Z 443.093,A -85,B 0,C 180,E1 -23305.046,E2 -23305.046} C_VEL
LIN {X 0,Y 162.483,Z 443.887,A -85,B 0,C 180,E1 -23307.52,E2 -23307.52} C_VEL
LIN {X 0,Y 162.385,Z 444.189,A -85,B 0,C 180,E1 -23309.999,E2 -23309.999} C_VEL
LIN {X 0,Y 162.479,Z 443.91,A -85,B 0,C 180,E1 -23312.478,E2 -23312.478} C_VEL
LIN {X 0,Y 162.799,Z 443.161,A -85,B 0,C 180,E1 -23314.952,E2 -23314.952} C_VEL
LIN {X 0,Y 163.341,Z 441.947,A -85,B 0,C 180,E1 -23317.415,E2 -23317.415} C_VEL
LIN {X 0,Y 164.463,Z 439.108,A -85,B 0,C 180,E1 -23321.086,E2 -23321.086} C_VEL
LIN {X 0,Y 165.466,Z 436.523,A -85,B 0,C 180,E1 -23323.508,E2 -23323.508} C_VEL
LIN {X 0,Y 167.418,Z 431.435,A -85,B 0,C 180,E1 -23327.087,E2 -23327.087} C_VEL
LIN {X 0,Y 169.555,Z 425.949,A -85,B 0,C 180,E1 -23329.995,E2 -23329.995} C_VEL
LIN {X 0,Y 172.051,Z 419.047,A -85,B 0,C 180,E1 -23332.832,E2 -23332.832} C_VEL
LIN {X 0,Y 174.416,Z 411.129,A -85,B 0,C 180,E1 -23335.347,E2 -23335.347} C_VEL
LIN {X 0,Y 176.55,Z 403.567,A -85,B 0,C 180,E1 -23337.243,E2 -23337.243} C_VEL
LIN {X 0,Y 178.562,Z 395.629,A -85,B 0,C 180,E1 -23338.824,E2 -23338.824} C_VEL
LIN {X 0,Y 180.241,Z 387.425,A -85,B 0,C 180,E1 -23340.133,E2 -23340.133} C_VEL
LIN {X 0,Y 181.625,Z 378.854,A -85,B 0,C 180,E1 -23341.199,E2 -23341.199} C_VEL
LIN {X 0,Y 182.569,Z 369.852,A -85,B 0,C 180,E1 -23342.06,E2 -23342.06} C_VEL
LIN {X 0,Y 183.277,Z 360.515,A -85,B 0,C 180,E1 -23342.653,E2 -23342.653} C_VEL
LIN {X 0,Y 184.549,Z 331.897,A -85,B 0,C 180,E1 -23343.758,E2 -23343.758} C_VEL
LIN {X 0,Y 177.991,Z 318.296,A -85,B 0,C 180,E1 -23345.865,E2 -23345.865} C_VEL
LIN {X 0,Y 171.086,Z 306.31,A -85,B 0,C 180,E1 -23348.206,E2 -23348.206} C_VEL
LIN {X 0,Y 167.006,Z 299.764,A -85,B 0,C 180,E1 -23349.69,E2 -23349.69} C_VEL
LIN {X 0,Y 164.894,Z 296.936,A -85,B 0,C 180,E1 -23350.47,E2 -23350.47} C_VEL
LIN {X 0,Y 164.285,Z 294.817,A -85,B 0,C 180,E1 -23350.835,E2 -23350.835} C_VEL
LIN {X 0,Y 164.277,Z 294.828,A -85,B 0,C 180,E1 -23353.341,E2 -23353.341} C_VEL
LIN {X 0,Y 164.256,Z 294.818,A -85,B 0,C 180,E1 -23356.796,E2 -23356.796} C_VEL
LIN {X 0,Y 164.286,Z 294.825,A -85,B 0,C 180,E1 -23360.354,E2 -23360.354} C_VEL
LIN {X 0,Y 164.322,Z 294.822,A -85,B 0,C 180,E1 -23364.35,E2 -23364.35} C_VEL
LIN {X 0,Y 164.363,Z 294.819,A -85,B 0,C 180,E1 -23369.129,E2 -23369.129} C_VEL
LIN {X 0,Y 164.39,Z 294.82,A -85,B 0,C 180,E1 -23374.689,E2 -23374.689} C_VEL
LIN {X 0,Y 164.413,Z 294.817,A -85,B 0,C 180,E1 -23380.117,E2 -23380.117} C_VEL
LIN {X 0,Y 164.467,Z 294.778,A -85,B 0,C 180,E1 -23385.144,E2 -23385.144} C_VEL
LIN {X 0,Y 164.759,Z 294.773,A -85,B 0,C 180,E1 -23390.176,E2 -23390.176} C_VEL
LIN {X 0,Y 164.813,Z 294.759,A -85,B 0,C 180,E1 -23392.65,E2 -23392.65} C_VEL
LIN {X 0,Y 165.269,Z 294.704,A -85,B 0,C 180,E1 -23400,E2 -23400} C_VEL
LIN {X 0,Y 164.815,Z 294.767,A -85,B 0,C 180,E1 -23407.349,E2 -23407.349} C_VEL
LIN {X 0,Y 164.697,Z 294.775,A -85,B 0,C 180,E1 -23411.057,E2 -23411.057} C_VEL
LIN {X 0,Y 164.424,Z 294.816,A -85,B 0,C 180,E1 -23417.409,E2 -23417.409} C_VEL
LIN {X 0,Y 164.415,Z 294.813,A -85,B 0,C 180,E1 -23419.996,E2 -23419.996} C_VEL
LIN {X 0,Y 164.334,Z 294.829,A -85,B 0,C 180,E1 -23426.095,E2 -23426.095} C_VEL
LIN {X 0,Y 164.353,Z 294.829,A -85,B 0,C 180,E1 -23431.217,E2 -23431.217} C_VEL
LIN {X 0,Y 164.275,Z 294.839,A -85,B 0,C 180,E1 -23436.794,E2 -23436.794} C_VEL
LIN {X 0,Y 164.281,Z 294.839,A -85,B 0,C 180,E1 -23439.919,E2 -23439.919} C_VEL
LIN {X 0,Y 164.274,Z 294.838,A -85,B 0,C 180,E1 -23445.609,E2 -23445.609} C_VEL
LIN {X 0,Y 165.521,Z 299.681,A -85,B 0,C 180,E1 -23449.14,E2 -23449.14} C_VEL
LIN {X 0,Y 167.665,Z 303.881,A -85,B 0,C 180,E1 -23449.992,E2 -23449.992} C_VEL
LIN {X 0,Y 171.408,Z 311.143,A -85,B 0,C 180,E1 -23451.401,E2 -23451.401} C_VEL
LIN {X 0,Y 176.599,Z 322.396,A -85,B 0,C 180,E1 -23453.275,E2 -23453.275} C_VEL
LIN {X 0,Y 180.308,Z 332.015,A -85,B 0,C 180,E1 -23454.597,E2 -23454.597} C_VEL
LIN {X 0,Y 182.884,Z 356.002,A -85,B 0,C 180,E1 -23456.273,E2 -23456.273} C_VEL
LIN {X 0,Y 183.21,Z 362.787,A -85,B 0,C 180,E1 -23456.651,E2 -23456.651} C_VEL
LIN {X 0,Y 182.217,Z 381.033,A -85,B 0,C 180,E1 -23457.402,E2 -23457.402} C_VEL
LIN {X 0,Y 180.734,Z 393.412,A -85,B 0,C 180,E1 -23458.336,E2 -23458.336} C_VEL
LIN {X 0,Y 179.07,Z 402.402,A -85,B 0,C 180,E1 -23459.323,E2 -23459.323} C_VEL
LIN {X 0,Y 177.18,Z 411.081,A -85,B 0,C 180,E1 -23460.604,E2 -23460.604} C_VEL
LIN {X 0,Y 174.95,Z 419.608,A -85,B 0,C 180,E1 -23462.223,E2 -23462.223} C_VEL
LIN {X 0,Y 172.747,Z 427.245,A -85,B 0,C 180,E1 -23464.067,E2 -23464.067} C_VEL
LIN {X 0,Y 170.318,Z 434.604,A -85,B 0,C 180,E1 -23466.278,E2 -23466.278} C_VEL
LIN {X 0,Y 167.82,Z 442.084,A -85,B 0,C 180,E1 -23469.149,E2 -23469.149} C_VEL
LIN {X 0,Y 165.313,Z 448.916,A -85,B 0,C 180,E1 -23472.688,E2 -23472.688} C_VEL
LIN {X 0,Y 164.374,Z 451.696,A -85,B 0,C 180,E1 -23474.485,E2 -23474.485} C_VEL
LIN {X 0,Y 162.944,Z 454.161,A -85,B 0,C 180,E1 -23476.304,E2 -23476.304} C_VEL
LIN {X 0,Y 160.732,Z 456.214,A -85,B 0,C 180,E1 -23478.123,E2 -23478.123} C_VEL
LIN {X 0,Y 157.542,Z 458.397,A -85,B 0,C 180,E1 -23480.637,E2 -23480.637} C_VEL
LIN {X 0,Y 155.19,Z 460.139,A -85,B 0,C 180,E1 -23483.532,E2 -23483.532} C_VEL
LIN {X 0,Y 154.919,Z 460.611,A -85,B 0,C 180,E1 -23484.783,E2 -23484.783} C_VEL
LIN {X 0,Y 154.953,Z 461.413,A -85,B 0,C 180,E1 -23487.402,E2 -23487.402} C_VEL
LIN {X 0,Y 155.188,Z 461.724,A -85,B 0,C 180,E1 -23490.001,E2 -23490.001} C_VEL
LIN {X 0,Y 154.922,Z 461.192,A -85,B 0,C 180,E1 -23493.609,E2 -23493.609} C_VEL
LIN {X 0,Y 155.062,Z 459.288,A -85,B 0,C 180,E1 -23497.816,E2 -23497.816} C_VEL
LIN {X 0,Y 155.831,Z 456.326,A -85,B 0,C 180,E1 -23501.711,E2 -23501.711} C_VEL
LIN {X 0,Y 156.664,Z 453.633,A -85,B 0,C 180,E1 -23504.286,E2 -23504.286} C_VEL
LIN {X 0,Y 158.523,Z 448.393,A -85,B 0,C 180,E1 -23508.081,E2 -23508.081} C_VEL
LIN {X 0,Y 161.194,Z 441.503,A -85,B 0,C 180,E1 -23511.754,E2 -23511.754} C_VEL
LIN {X 0,Y 163.835,Z 433.985,A -85,B 0,C 180,E1 -23514.725,E2 -23514.725} C_VEL
LIN {X 0,Y 166.425,Z 426.588,A -85,B 0,C 180,E1 -23517,E2 -23517} C_VEL
LIN {X 0,Y 168.434,Z 419.8,A -85,B 0,C 180,E1 -23518.702,E2 -23518.702} C_VEL
LIN {X 0,Y 170.591,Z 411.785,A -85,B 0,C 180,E1 -23520.311,E2 -23520.311} C_VEL
LIN {X 0,Y 172.572,Z 403.38,A -85,B 0,C 180,E1 -23521.625,E2 -23521.625} C_VEL
LIN {X 0,Y 174.263,Z 394.787,A -85,B 0,C 180,E1 -23522.645,E2 -23522.645} C_VEL
LIN {X 0,Y 175.684,Z 385.345,A -85,B 0,C 180,E1 -23523.457,E2 -23523.457} C_VEL
LIN {X 0,Y 176.645,Z 374.123,A -85,B 0,C 180,E1 -23524.101,E2 -23524.101} C_VEL
LIN {X 0,Y 177.2,Z 361.388,A -85,B 0,C 180,E1 -23524.594,E2 -23524.594} C_VEL
LIN {X 0,Y 174.705,Z 335.447,A -85,B 0,C 180,E1 -23526.433,E2 -23526.433} C_VEL
LIN {X 0,Y 173.898,Z 332.34,A -85,B 0,C 180,E1 -23526.783,E2 -23526.783} C_VEL
LIN {X 0,Y 168.699,Z 319.671,A -85,B 0,C 180,E1 -23528.765,E2 -23528.765} C_VEL
LIN {X 0,Y 163.296,Z 308.695,A -85,B 0,C 180,E1 -23530.9,E2 -23530.9} C_VEL
LIN {X 0,Y 160.234,Z 303.233,A -85,B 0,C 180,E1 -23532.162,E2 -23532.162} C_VEL
LIN {X 0,Y 158.029,Z 298.895,A -85,B 0,C 180,E1 -23533.233,E2 -23533.233} C_VEL
LIN {X 0,Y 157.217,Z 295.717,A -85,B 0,C 180,E1 -23535.87,E2 -23535.87} C_VEL
LIN {X 0,Y 157.199,Z 295.72,A -85,B 0,C 180,E1 -23541.252,E2 -23541.252} C_VEL
LIN {X 0,Y 157.276,Z 295.711,A -85,B 0,C 180,E1 -23544.485,E2 -23544.485} C_VEL
LIN {X 0,Y 157.277,Z 295.705,A -85,B 0,C 180,E1 -23548.108,E2 -23548.108} C_VEL
LIN {X 0,Y 157.268,Z 295.709,A -85,B 0,C 180,E1 -23553.457,E2 -23553.457} C_VEL
LIN {X 0,Y 157.362,Z 295.692,A -85,B 0,C 180,E1 -23559.703,E2 -23559.703} C_VEL
LIN {X 0,Y 157.406,Z 295.686,A -85,B 0,C 180,E1 -23564.461,E2 -23564.461} C_VEL
LIN {X 0,Y 157.687,Z 295.632,A -85,B 0,C 180,E1 -23569.731,E2 -23569.731} C_VEL
LIN {X 0,Y 157.757,Z 295.608,A -85,B 0,C 180,E1 -23572.32,E2 -23572.32} C_VEL
LIN {X 0,Y 158.238,Z 295.579,A -85,B 0,C 180,E1 -23580,E2 -23580} C_VEL
LIN {X 0,Y 157.759,Z 295.64,A -85,B 0,C 180,E1 -23587.681,E2 -23587.681} C_VEL
LIN {X 0,Y 157.633,Z 295.656,A -85,B 0,C 180,E1 -23591.223,E2 -23591.223} C_VEL
LIN {X 0,Y 157.405,Z 295.655,A -85,B 0,C 180,E1 -23595.539,E2 -23595.539} C_VEL
LIN {X 0,Y 157.306,Z 295.703,A -85,B 0,C 180,E1 -23600.942,E2 -23600.942} C_VEL
LIN {X 0,Y 157.269,Z 295.704,A -85,B 0,C 180,E1 -23606.649,E2 -23606.649} C_VEL
LIN {X 0,Y 157.271,Z 295.697,A -85,B 0,C 180,E1 -23612.429,E2 -23612.429} C_VEL
LIN {X 0,Y 157.261,Z 295.689,A -85,B 0,C 180,E1 -23616.444,E2 -23616.444} C_VEL
LIN {X 0,Y 157.191,Z 295.7,A -85,B 0,C 180,E1 -23622.118,E2 -23622.118} C_VEL
LIN {X 0,Y 157.244,Z 295.782,A -85,B 0,C 180,E1 -23627.225,E2 -23627.225} C_VEL
LIN {X 0,Y 158.084,Z 298.33,A -85,B 0,C 180,E1 -23627.664,E2 -23627.664} C_VEL
LIN {X 0,Y 160.224,Z 300.991,A -85,B 0,C 180,E1 -23628.525,E2 -23628.525} C_VEL
LIN {X 0,Y 162.546,Z 304.513,A -85,B 0,C 180,E1 -23629.457,E2 -23629.457} C_VEL
LIN {X 0,Y 169.228,Z 315.482,A -85,B 0,C 180,E1 -23631.977,E2 -23631.977} C_VEL
LIN {X 0,Y 175.519,Z 327.321,A -85,B 0,C 180,E1 -23634.179,E2 -23634.179} C_VEL
LIN {X 0,Y 178.57,Z 333.908,A -85,B 0,C 180,E1 -23635.211,E2 -23635.211} C_VEL
LIN {X 0,Y 177.2,Z 361.03,A -85,B 0,C 180,E1 -23636.27,E2 -23636.27} C_VEL
LIN {X 0,Y 176.398,Z 370.51,A -85,B 0,C 180,E1 -23636.886,E2 -23636.886} C_VEL
LIN {X 0,Y 175.544,Z 378.318,A -85,B 0,C 180,E1 -23637.642,E2 -23637.642} C_VEL
LIN {X 0,Y 174.227,Z 386.799,A -85,B 0,C 180,E1 -23638.71,E2 -23638.71} C_VEL
LIN {X 0,Y 172.406,Z 395.208,A -85,B 0,C 180,E1 -23640.041,E2 -23640.041} C_VEL
LIN {X 0,Y 170.65,Z 402.069,A -85,B 0,C 180,E1 -23641.394,E2 -23641.394} C_VEL
LIN {X 0,Y 168.696,Z 408.94,A -85,B 0,C 180,E1 -23643.058,E2 -23643.058} C_VEL
LIN {X 0,Y 166.726,Z 415.606,A -85,B 0,C 180,E1 -23645.068,E2 -23645.068} C_VEL
LIN {X 0,Y 164.509,Z 421.926,A -85,B 0,C 180,E1 -23647.387,E2 -23647.387} C_VEL
LIN {X 0,Y 162.483,Z 427.178,A -85,B 0,C 180,E1 -23649.754,E2 -23649.754} C_VEL
LIN {X 0,Y 160.716,Z 431.56,A -85,B 0,C 180,E1 -23652.174,E2 -23652.174} C_VEL
LIN {X 0,Y 158.62,Z 436.705,A -85,B 0,C 180,E1 -23655.894,E2 -23655.894} C_VEL
LIN {X 0,Y 157.508,Z 439.343,A -85,B 0,C 180,E1 -23658.416,E2 -23658.416} C_VEL
LIN {X 0,Y 157.014,Z 440.73,A -85,B 0,C 180,E1 -23659.976,E2 -23659.976} C_VEL
LIN {X 0,Y 156.339,Z 442.226,A -85,B 0,C 180,E1 -23662.248,E2 -23662.248} C_VEL
LIN {X 0,Y 155.774,Z 443.485,A -85,B 0,C 180,E1 -23664.822,E2 -23664.822} C_VEL
LIN {X 0,Y 155.411,Z 444.278,A -85,B 0,C 180,E1 -23667.407,E2 -23667.407} C_VEL
LIN {X 0,Y 155.305,Z 444.58,A -85,B 0,C 180,E1 -23669.999,E2 -23669.999} C_VEL
LIN {X 0,Y 155.406,Z 444.3,A -85,B 0,C 180,E1 -23672.591,E2 -23672.591} C_VEL
LIN {X 0,Y 155.75,Z 443.552,A -85,B 0,C 180,E1 -23675.176,E2 -23675.176} C_VEL
LIN {X 0,Y 156.31,Z 442.338,A -85,B 0,C 180,E1 -23677.751,E2 -23677.751} C_VEL
LIN {X 0,Y 157.091,Z 440.636,A -85,B 0,C 180,E1 -23680.307,E2 -23680.307} C_VEL
LIN {X 0,Y 158.594,Z 436.912,A -85,B 0,C 180,E1 -23684.105,E2 -23684.105} C_VEL
LIN {X 0,Y 160.661,Z 431.824,A -85,B 0,C 180,E1 -23687.83,E2 -23687.83} C_VEL
LIN {X 0,Y 162.924,Z 426.338,A -85,B 0,C 180,E1 -23690.846,E2 -23690.846} C_VEL
LIN {X 0,Y 165.555,Z 419.435,A -85,B 0,C 180,E1 -23693.782,E2 -23693.782} C_VEL
LIN {X 0,Y 168.028,Z 411.517,A -85,B 0,C 180,E1 -23696.384,E2 -23696.384} C_VEL
LIN {X 0,Y 170.299,Z 403.953,A -85,B 0,C 180,E1 -23698.331,E2 -23698.331} C_VEL
LIN {X 0,Y 172.386,Z 396.016,A -85,B 0,C 180,E1 -23699.96,E2 -23699.96} C_VEL
LIN {X 0,Y 174.158,Z 387.81,A -85,B 0,C 180,E1 -23701.301,E2 -23701.301} C_VEL
LIN {X 0,Y 175.705,Z 378.554,A -85,B 0,C 180,E1 -23702.471,E2 -23702.471} C_VEL
LIN {X 0,Y 176.819,Z 368.15,A -85,B 0,C 180,E1 -23703.448,E2 -23703.448} C_VEL
LIN {X 0,Y 177.709,Z 354.141,A -85,B 0,C 180,E1 -23704.19,E2 -23704.19} C_VEL
LIN {X 0,Y 178.623,Z 334.045,A -85,B 0,C 180,E1 -23704.953,E2 -23704.953} C_VEL
LIN {X 0,Y 172.28,Z 320.872,A -85,B 0,C 180,E1 -23707.137,E2 -23707.137} C_VEL
LIN {X 0,Y 164.816,Z 308.105,A -85,B 0,C 180,E1 -23709.866,E2 -23709.866} C_VEL
LIN {X 0,Y 160.195,Z 300.955,A -85,B 0,C 180,E1 -23711.7,E2 -23711.7} C_VEL
LIN {X 0,Y 157.81,Z 297.778,A -85,B 0,C 180,E1 -23712.68,E2 -23712.68} C_VEL
LIN {X 0,Y 157.213,Z 295.704,A -85,B 0,C 180,E1 -23713.082,E2 -23713.082} C_VEL
LIN {X 0,Y 157.186,Z 295.693,A -85,B 0,C 180,E1 -23717.881,E2 -23717.881} C_VEL
LIN {X 0,Y 157.255,Z 295.7,A -85,B 0,C 180,E1 -23723.555,E2 -23723.555} C_VEL
LIN {X 0,Y 157.276,Z 295.698,A -85,B 0,C 180,E1 -23728.103,E2 -23728.103} C_VEL
LIN {X 0,Y 157.306,Z 295.697,A -85,B 0,C 180,E1 -23733.463,E2 -23733.463} C_VEL
LIN {X 0,Y 157.356,Z 295.697,A -85,B 0,C 180,E1 -23739.701,E2 -23739.701} C_VEL
LIN {X 0,Y 157.401,Z 295.658,A -85,B 0,C 180,E1 -23744.46,E2 -23744.46} C_VEL
LIN {X 0,Y 157.682,Z 295.655,A -85,B 0,C 180,E1 -23749.73,E2 -23749.73} C_VEL
LIN {X 0,Y 157.752,Z 295.641,A -85,B 0,C 180,E1 -23752.319,E2 -23752.319} C_VEL
LIN {X 0,Y 158.231,Z 295.581,A -85,B 0,C 180,E1 -23760,E2 -23760} C_VEL
LIN {X 0,Y 157.754,Z 295.647,A -85,B 0,C 180,E1 -23767.68,E2 -23767.68} C_VEL
LIN {X 0,Y 157.626,Z 295.656,A -85,B 0,C 180,E1 -23771.223,E2 -23771.223} C_VEL
LIN {X 0,Y 157.401,Z 295.686,A -85,B 0,C 180,E1 -23775.539,E2 -23775.539} C_VEL
LIN {X 0,Y 157.299,Z 295.701,A -85,B 0,C 180,E1 -23780.942,E2 -23780.942} C_VEL
LIN {X 0,Y 157.262,Z 295.711,A -85,B 0,C 180,E1 -23786.649,E2 -23786.649} C_VEL
LIN {X 0,Y 157.264,Z 295.712,A -85,B 0,C 180,E1 -23792.43,E2 -23792.43} C_VEL
LIN {X 0,Y 157.254,Z 295.714,A -85,B 0,C 180,E1 -23796.445,E2 -23796.445} C_VEL
LIN {X 0,Y 157.186,Z 295.722,A -85,B 0,C 180,E1 -23802.119,E2 -23802.119} C_VEL
LIN {X 0,Y 157.228,Z 295.722,A -85,B 0,C 180,E1 -23804.126,E2 -23804.126} C_VEL
LIN {X 0,Y 158.173,Z 299.307,A -85,B 0,C 180,E1 -23806.804,E2 -23806.804} C_VEL
LIN {X 0,Y 160.302,Z 303.361,A -85,B 0,C 180,E1 -23807.744,E2 -23807.744} C_VEL
LIN {X 0,Y 161.696,Z 305.829,A -85,B 0,C 180,E1 -23808.329,E2 -23808.329} C_VEL
LIN {X 0,Y 166.078,Z 314.043,A -85,B 0,C 180,E1 -23810.097,E2 -23810.097} C_VEL
LIN {X 0,Y 171.894,Z 327.045,A -85,B 0,C 180,E1 -23812.351,E2 -23812.351} C_VEL
LIN {X 0,Y 174.769,Z 334.993,A -85,B 0,C 180,E1 -23813.462,E2 -23813.462} C_VEL
LIN {X 0,Y 177.135,Z 358.859,A -85,B 0,C 180,E1 -23815.178,E2 -23815.178} C_VEL
LIN {X 0,Y 177.26,Z 363.675,A -85,B 0,C 180,E1 -23815.437,E2 -23815.437} C_VEL
LIN {X 0,Y 176.286,Z 380.657,A -85,B 0,C 180,E1 -23816.16,E2 -23816.16} C_VEL
LIN {X 0,Y 174.74,Z 393.028,A -85,B 0,C 180,E1 -23817.116,E2 -23817.116} C_VEL
LIN {X 0,Y 172.999,Z 402.016,A -85,B 0,C 180,E1 -23818.123,E2 -23818.123} C_VEL
LIN {X 0,Y 171.029,Z 410.693,A -85,B 0,C 180,E1 -23819.436,E2 -23819.436} C_VEL
LIN {X 0,Y 168.958,Z 418.271,A -85,B 0,C 180,E1 -23820.885,E2 -23820.885} C_VEL
LIN {X 0,Y 166.718,Z 425.831,A -85,B 0,C 180,E1 -23822.715,E2 -23822.715} C_VEL
LIN {X 0,Y 164.464,Z 432.503,A -85,B 0,C 180,E1 -23824.704,E2 -23824.704} C_VEL
LIN {X 0,Y 162.193,Z 438.846,A -85,B 0,C 180,E1 -23827.048,E2 -23827.048} C_VEL
LIN {X 0,Y 160.224,Z 444.121,A -85,B 0,C 180,E1 -23829.459,E2 -23829.459} C_VEL
LIN {X 0,Y 158.524,Z 448.524,A -85,B 0,C 180,E1 -23831.922,E2 -23831.922} C_VEL
LIN {X 0,Y 156.674,Z 453.736,A -85,B 0,C 180,E1 -23835.718,E2 -23835.718} C_VEL
LIN {X 0,Y 155.51,Z 457.575,A -85,B 0,C 180,E1 -23839.587,E2 -23839.587} C_VEL
LIN {X 0,Y 155.061,Z 459.343,A -85,B 0,C 180,E1 -23842.187,E2 -23842.187} C_VEL
LIN {X 0,Y 154.919,Z 460.611,A -85,B 0,C 180,E1 -23844.783,E2 -23844.783} C_VEL
LIN {X 0,Y 154.241,Z 461.382,A -85,B 0,C 180,E1 -23846.935,E2 -23846.935} C_VEL
LIN {X 0,Y 152.632,Z 461.647,A -85,B 0,C 180,E1 -23849.073,E2 -23849.073} C_VEL
LIN {X 0,Y 148.902,Z 460.95,A -85,B 0,C 180,E1 -23853.435,E2 -23853.435} C_VEL
LIN {X 0,Y 147.916,Z 460.101,A -85,B 0,C 180,E1 -23855.714,E2 -23855.714} C_VEL
LIN {X 0,Y 147.867,Z 459.706,A -85,B 0,C 180,E1 -23856.483,E2 -23856.483} C_VEL
LIN {X 0,Y 148.52,Z 457.103,A -85,B 0,C 180,E1 -23860.912,E2 -23860.912} C_VEL
LIN {X 0,Y 149.257,Z 454.739,A -85,B 0,C 180,E1 -23863.618,E2 -23863.618} C_VEL
LIN {X 0,Y 151.013,Z 449.931,A -85,B 0,C 180,E1 -23867.609,E2 -23867.609} C_VEL
LIN {X 0,Y 153.094,Z 444.745,A -85,B 0,C 180,E1 -23870.842,E2 -23870.842} C_VEL
LIN {X 0,Y 155.129,Z 439.683,A -85,B 0,C 180,E1 -23873.355,E2 -23873.355} C_VEL
LIN {X 0,Y 157.419,Z 433.591,A -85,B 0,C 180,E1 -23875.805,E2 -23875.805} C_VEL
LIN {X 0,Y 160.132,Z 426.193,A -85,B 0,C 180,E1 -23878.153,E2 -23878.153} C_VEL
LIN {X 0,Y 162.276,Z 419.244,A -85,B 0,C 180,E1 -23879.946,E2 -23879.946} C_VEL
LIN {X 0,Y 164.492,Z 411.388,A -85,B 0,C 180,E1 -23881.561,E2 -23881.561} C_VEL
LIN {X 0,Y 166.557,Z 402.982,A -85,B 0,C 180,E1 -23882.908,E2 -23882.908} C_VEL
LIN {X 0,Y 168.288,Z 394.673,A -85,B 0,C 180,E1 -23883.915,E2 -23883.915} C_VEL
LIN {X 0,Y 169.824,Z 384.959,A -85,B 0,C 180,E1 -23884.772,E2 -23884.772} C_VEL
LIN {X 0,Y 170.824,Z 373.528,A -85,B 0,C 180,E1 -23885.444,E2 -23885.444} C_VEL
LIN {X 0,Y 171.337,Z 362.005,A -85,B 0,C 180,E1 -23885.906,E2 -23885.906} C_VEL
LIN {X 0,Y 169.098,Z 337.415,A -85,B 0,C 180,E1 -23887.724,E2 -23887.724} C_VEL
LIN {X 0,Y 166.683,Z 330.417,A -85,B 0,C 180,E1 -23888.735,E2 -23888.735} C_VEL
LIN {X 0,Y 161.925,Z 319.534,A -85,B 0,C 180,E1 -23890.695,E2 -23890.695} C_VEL
LIN {X 0,Y 157.652,Z 311.149,A -85,B 0,C 180,E1 -23892.527,E2 -23892.527} C_VEL
LIN {X 0,Y 155.644,Z 307.523,A -85,B 0,C 180,E1 -23893.423,E2 -23893.423} C_VEL
LIN {X 0,Y 153.159,Z 303.069,A -85,B 0,C 180,E1 -23894.581,E2 -23894.581} C_VEL
LIN {X 0,Y 150.784,Z 298.789,A -85,B 0,C 180,E1 -23895.748,E2 -23895.748} C_VEL
LIN {X 0,Y 150.459,Z 297.848,A -85,B 0,C 180,E1 -23896.366,E2 -23896.366} C_VEL
LIN {X 0,Y 150.169,Z 296.595,A -85,B 0,C 180,E1 -23897.51,E2 -23897.51} C_VEL
LIN {X 0,Y 150.177,Z 296.595,A -85,B 0,C 180,E1 -23902.711,E2 -23902.711} C_VEL
LIN {X 0,Y 150.204,Z 296.587,A -85,B 0,C 180,E1 -23907.377,E2 -23907.377} C_VEL
LIN {X 0,Y 150.184,Z 296.59,A -85,B 0,C 180,E1 -23912.766,E2 -23912.766} C_VEL
LIN {X 0,Y 150.284,Z 296.574,A -85,B 0,C 180,E1 -23919.279,E2 -23919.279} C_VEL
LIN {X 0,Y 150.312,Z 296.57,A -85,B 0,C 180,E1 -23923.708,E2 -23923.708} C_VEL
LIN {X 0,Y 150.607,Z 296.519,A -85,B 0,C 180,E1 -23929.243,E2 -23929.243} C_VEL
LIN {X 0,Y 150.68,Z 296.488,A -85,B 0,C 180,E1 -23931.957,E2 -23931.957} C_VEL
LIN {X 0,Y 151.198,Z 296.455,A -85,B 0,C 180,E1 -23940,E2 -23940} C_VEL
LIN {X 0,Y 150.698,Z 296.522,A -85,B 0,C 180,E1 -23948.043,E2 -23948.043} C_VEL
LIN {X 0,Y 150.576,Z 296.534,A -85,B 0,C 180,E1 -23951.427,E2 -23951.427} C_VEL
LIN {X 0,Y 150.31,Z 296.541,A -85,B 0,C 180,E1 -23956.293,E2 -23956.293} C_VEL
LIN {X 0,Y 150.284,Z 296.578,A -85,B 0,C 180,E1 -23960.721,E2 -23960.721} C_VEL
LIN {X 0,Y 150.187,Z 296.584,A -85,B 0,C 180,E1 -23967.237,E2 -23967.237} C_VEL
LIN {X 0,Y 150.211,Z 296.573,A -85,B 0,C 180,E1 -23972.627,E2 -23972.627} C_VEL
LIN {X 0,Y 150.172,Z 296.583,A -85,B 0,C 180,E1 -23977.474,E2 -23977.474} C_VEL
LIN {X 0,Y 150.134,Z 296.581,A -85,B 0,C 180,E1 -23981.496,E2 -23981.496} C_VEL
LIN {X 0,Y 150.13,Z 296.61,A -85,B 0,C 180,E1 -23984.675,E2 -23984.675} C_VEL
LIN {X 0,Y 151.071,Z 299.348,A -85,B 0,C 180,E1 -23985.221,E2 -23985.221} C_VEL
LIN {X 0,Y 153.357,Z 302.028,A -85,B 0,C 180,E1 -23986.246,E2 -23986.246} C_VEL
LIN {X 0,Y 155.56,Z 305.364,A -85,B 0,C 180,E1 -23987.236,E2 -23987.236} C_VEL
LIN {X 0,Y 161.918,Z 315.307,A -85,B 0,C 180,E1 -23989.883,E2 -23989.883} C_VEL
LIN {X 0,Y 168.67,Z 327.51,A -85,B 0,C 180,E1 -23992.465,E2 -23992.465} C_VEL
LIN {X 0,Y 172.706,Z 336.031,A -85,B 0,C 180,E1 -23993.935,E2 -23993.935} C_VEL
LIN {X 0,Y 171.352,Z 361.438,A -85,B 0,C 180,E1 -23994.954,E2 -23994.954} C_VEL
LIN {X 0,Y 170.493,Z 371.049,A -85,B 0,C 180,E1 -23995.596,E2 -23995.596} C_VEL
LIN {X 0,Y 169.493,Z 379.655,A -85,B 0,C 180,E1 -23996.476,E2 -23996.476} C_VEL
LIN {X 0,Y 167.858,Z 389.061,A -85,B 0,C 180,E1 -23997.734,E2 -23997.734} C_VEL
LIN {X 0,Y 165.545,Z 398.595,A -85,B 0,C 180,E1 -23999.372,E2 -23999.372} C_VEL
LIN {X 0,Y 162.746,Z 408.319,A -85,B 0,C 180,E1 -24001.638,E2 -24001.638} C_VEL
LIN {X 0,Y 160.342,Z 415.999,A -85,B 0,C 180,E1 -24004.002,E2 -24004.002} C_VEL
LIN {X 0,Y 158.005,Z 422.318,A -85,B 0,C 180,E1 -24006.401,E2 -24006.401} C_VEL
LIN {X 0,Y 155.872,Z 427.57,A -85,B 0,C 180,E1 -24008.855,E2 -24008.855} C_VEL
LIN {X 0,Y 153.995,Z 431.952,A -85,B 0,C 180,E1 -24011.368,E2 -24011.368} C_VEL
LIN {X 0,Y 151.768,Z 437.097,A -85,B 0,C 180,E1 -24015.243,E2 -24015.243} C_VEL
LIN {X 0,Y 150.571,Z 439.735,A -85,B 0,C 180,E1 -24017.874,E2 -24017.874} C_VEL
LIN {X 0,Y 149.894,Z 441.447,A -85,B 0,C 180,E1 -24019.939,E2 -24019.939} C_VEL
LIN {X 0,Y 148.729,Z 443.876,A -85,B 0,C 180,E1 -24024.576,E2 -24024.576} C_VEL
LIN {X 0,Y 148.341,Z 444.669,A -85,B 0,C 180,E1 -24027.283,E2 -24027.283} C_VEL
LIN {X 0,Y 148.227,Z 444.971,A -85,B 0,C 180,E1 -24029.999,E2 -24029.999} C_VEL
LIN {X 0,Y 148.337,Z 444.691,A -85,B 0,C 180,E1 -24032.714,E2 -24032.714} C_VEL
LIN {X 0,Y 148.705,Z 443.942,A -85,B 0,C 180,E1 -24035.422,E2 -24035.422} C_VEL
LIN {X 0,Y 149.953,Z 441.48,A -85,B 0,C 180,E1 -24040.189,E2 -24040.189} C_VEL
LIN {X 0,Y 151.122,Z 438.744,A -85,B 0,C 180,E1 -24043.444,E2 -24043.444} C_VEL
LIN {X 0,Y 153.132,Z 434.108,A -85,B 0,C 180,E1 -24047.355,E2 -24047.355} C_VEL
LIN {X 0,Y 155.316,Z 429.056,A -85,B 0,C 180,E1 -24050.528,E2 -24050.528} C_VEL
LIN {X 0,Y 157.347,Z 424.115,A -85,B 0,C 180,E1 -24053.004,E2 -24053.004} C_VEL
LIN {X 0,Y 159.655,Z 418.147,A -85,B 0,C 180,E1 -24055.415,E2 -24055.415} C_VEL
LIN {X 0,Y 162.023,Z 410.891,A -85,B 0,C 180,E1 -24057.793,E2 -24057.793} C_VEL
LIN {X 0,Y 164.106,Z 404.34,A -85,B 0,C 180,E1 -24059.503,E2 -24059.503} C_VEL
LIN {X 0,Y 166.295,Z 396.402,A -85,B 0,C 180,E1 -24061.177,E2 -24061.177} C_VEL
LIN {X 0,Y 168.154,Z 388.194,A -85,B 0,C 180,E1 -24062.553,E2 -24062.553} C_VEL
LIN {X 0,Y 169.707,Z 379.422,A -85,B 0,C 180,E1 -24063.698,E2 -24063.698} C_VEL
LIN {X 0,Y 170.811,Z 370.066,A -85,B 0,C 180,E1 -24064.624,E2 -24064.624} C_VEL
LIN {X 0,Y 171.61,Z 360.311,A -85,B 0,C 180,E1 -24065.251,E2 -24065.251} C_VEL
LIN {X 0,Y 172.883,Z 336.418,A -85,B 0,C 180,E1 -24066.192,E2 -24066.192} C_VEL
LIN {X 0,Y 167.112,Z 324.456,A -85,B 0,C 180,E1 -24068.316,E2 -24068.316} C_VEL
LIN {X 0,Y 160.551,Z 313.03,A -85,B 0,C 180,E1 -24070.878,E2 -24070.878} C_VEL
LIN {X 0,Y 155.248,Z 305.032,A -85,B 0,C 180,E1 -24073.115,E2 -24073.115} C_VEL
LIN {X 0,Y 152.791,Z 301.297,A -85,B 0,C 180,E1 -24074.236,E2 -24074.236} C_VEL
LIN {X 0,Y 150.802,Z 298.86,A -85,B 0,C 180,E1 -24075.148,E2 -24075.148} C_VEL
LIN {X 0,Y 150.15,Z 296.584,A -85,B 0,C 180,E1 -24075.617,E2 -24075.617} C_VEL
LIN {X 0,Y 150.132,Z 296.575,A -85,B 0,C 180,E1 -24079.052,E2 -24079.052} C_VEL
LIN {X 0,Y 150.172,Z 296.584,A -85,B 0,C 180,E1 -24082.709,E2 -24082.709} C_VEL
LIN {X 0,Y 150.202,Z 296.579,A -85,B 0,C 180,E1 -24087.373,E2 -24087.373} C_VEL
LIN {X 0,Y 150.235,Z 296.575,A -85,B 0,C 180,E1 -24092.722,E2 -24092.722} C_VEL
LIN {X 0,Y 150.28,Z 296.577,A -85,B 0,C 180,E1 -24099.275,E2 -24099.275} C_VEL
LIN {X 0,Y 150.306,Z 296.545,A -85,B 0,C 180,E1 -24103.707,E2 -24103.707} C_VEL
LIN {X 0,Y 150.602,Z 296.533,A -85,B 0,C 180,E1 -24109.241,E2 -24109.241} C_VEL
LIN {X 0,Y 150.691,Z 296.523,A -85,B 0,C 180,E1 -24111.957,E2 -24111.957} C_VEL
LIN {X 0,Y 151.192,Z 296.457,A -85,B 0,C 180,E1 -24120,E2 -24120} C_VEL
LIN {X 0,Y 150.693,Z 296.527,A -85,B 0,C 180,E1 -24128.043,E2 -24128.043} C_VEL
LIN {X 0,Y 150.569,Z 296.535,A -85,B 0,C 180,E1 -24131.428,E2 -24131.428} C_VEL
LIN {X 0,Y 150.307,Z 296.57,A -85,B 0,C 180,E1 -24136.293,E2 -24136.293} C_VEL
LIN {X 0,Y 150.278,Z 296.574,A -85,B 0,C 180,E1 -24140.722,E2 -24140.722} C_VEL
LIN {X 0,Y 150.18,Z 296.594,A -85,B 0,C 180,E1 -24147.238,E2 -24147.238} C_VEL
LIN {X 0,Y 150.204,Z 296.591,A -85,B 0,C 180,E1 -24152.628,E2 -24152.628} C_VEL
LIN {X 0,Y 150.165,Z 296.596,A -85,B 0,C 180,E1 -24157.475,E2 -24157.475} C_VEL
LIN {X 0,Y 150.162,Z 296.689,A -85,B 0,C 180,E1 -24162.493,E2 -24162.493} C_VEL
LIN {X 0,Y 150.714,Z 298.573,A -85,B 0,C 180,E1 -24164.067,E2 -24164.067} C_VEL
LIN {X 0,Y 152.921,Z 302.737,A -85,B 0,C 180,E1 -24165.173,E2 -24165.173} C_VEL
LIN {X 0,Y 154.33,Z 305.131,A -85,B 0,C 180,E1 -24165.835,E2 -24165.835} C_VEL
LIN {X 0,Y 157.441,Z 310.709,A -85,B 0,C 180,E1 -24167.25,E2 -24167.25} C_VEL
LIN {X 0,Y 161.306,Z 318.126,A -85,B 0,C 180,E1 -24168.919,E2 -24168.919} C_VEL
LIN {X 0,Y 166.558,Z 329.998,A -85,B 0,C 180,E1 -24171.1,E2 -24171.1} C_VEL
LIN {X 0,Y 169.219,Z 337.352,A -85,B 0,C 180,E1 -24172.2,E2 -24172.2} C_VEL
LIN {X 0,Y 171.459,Z 362.168,A -85,B 0,C 180,E1 -24174.033,E2 -24174.033} C_VEL
LIN {X 0,Y 170.456,Z 380.024,A -85,B 0,C 180,E1 -24174.818,E2 -24174.818} C_VEL
LIN {X 0,Y 168.788,Z 392.724,A -85,B 0,C 180,E1 -24175.812,E2 -24175.812} C_VEL
LIN {X 0,Y 167.026,Z 401.631,A -85,B 0,C 180,E1 -24176.84,E2 -24176.84} C_VEL
LIN {X 0,Y 164.943,Z 410.305,A -85,B 0,C 180,E1 -24178.18,E2 -24178.18} C_VEL
LIN {X 0,Y 162.596,Z 418.547,A -85,B 0,C 180,E1 -24179.822,E2 -24179.822} C_VEL
LIN {X 0,Y 160.091,Z 426.467,A -85,B 0,C 180,E1 -24181.842,E2 -24181.842} C_VEL
LIN {X 0,Y 157.42,Z 433.825,A -85,B 0,C 180,E1 -24184.198,E2 -24184.198} C_VEL
LIN {X 0,Y 154.627,Z 441.304,A -85,B 0,C 180,E1 -24187.275,E2 -24187.275} C_VEL
LIN {X 0,Y 151.772,Z 448.133,A -85,B 0,C 180,E1 -24191.088,E2 -24191.088} C_VEL
LIN {X 0,Y 149.774,Z 453.343,A -85,B 0,C 180,E1 -24195.045,E2 -24195.045} C_VEL
LIN {X 0,Y 148.519,Z 457.183,A -85,B 0,C 180,E1 -24199.091,E2 -24199.091} C_VEL
LIN {X 0,Y 148.011,Z 458.951,A -85,B 0,C 180,E1 -24201.812,E2 -24201.812} C_VEL
LIN {X 0,Y 147.838,Z 460.936,A -85,B 0,C 180,E1 -24206.662,E2 -24206.662} C_VEL
LIN {X 0,Y 148.103,Z 461.332,A -85,B 0,C 180,E1 -24210.001,E2 -24210.001} C_VEL
LIN {X 0,Y 147.838,Z 460.919,A -85,B 0,C 180,E1 -24213.339,E2 -24213.339} C_VEL
LIN {X 0,Y 147.867,Z 459.706,A -85,B 0,C 180,E1 -24216.483,E2 -24216.483} C_VEL
LIN {X 0,Y 147.398,Z 458.581,A -85,B 0,C 180,E1 -24218.722,E2 -24218.722} C_VEL
LIN {X 0,Y 146.192,Z 457.111,A -85,B 0,C 180,E1 -24220.923,E2 -24220.923} C_VEL
LIN {X 0,Y 144.42,Z 454.688,A -85,B 0,C 180,E1 -24223.835,E2 -24223.835} C_VEL
LIN {X 0,Y 143.653,Z 451.666,A -85,B 0,C 180,E1 -24226.743,E2 -24226.743} C_VEL
LIN {X 0,Y 144.07,Z 449.94,A -85,B 0,C 180,E1 -24228.152,E2 -24228.152} C_VEL
LIN {X 0,Y 146.001,Z 445.533,A -85,B 0,C 180,E1 -24231.165,E2 -24231.165} C_VEL
LIN {X 0,Y 148.591,Z 439.286,A -85,B 0,C 180,E1 -24234.449,E2 -24234.449} C_VEL
LIN {X 0,Y 151.068,Z 433.197,A -85,B 0,C 180,E1 -24236.976,E2 -24236.976} C_VEL
LIN {X 0,Y 153.901,Z 425.797,A -85,B 0,C 180,E1 -24239.402,E2 -24239.402} C_VEL
LIN {X 0,Y 156.387,Z 418.206,A -85,B 0,C 180,E1 -24241.393,E2 -24241.393} C_VEL
LIN {X 0,Y 158.924,Z 409.488,A -85,B 0,C 180,E1 -24243.18,E2 -24243.18} C_VEL
LIN {X 0,Y 161.511,Z 398.938,A -85,B 0,C 180,E1 -24244.799,E2 -24244.799} C_VEL
LIN {X 0,Y 163.619,Z 387.777,A -85,B 0,C 180,E1 -24245.927,E2 -24245.927} C_VEL
LIN {X 0,Y 164.657,Z 378.438,A -85,B 0,C 180,E1 -24246.599,E2 -24246.599} C_VEL
LIN {X 0,Y 165.601,Z 363.018,A -85,B 0,C 180,E1 -24247.28,E2 -24247.28} C_VEL
LIN {X 0,Y 163.584,Z 339.366,A -85,B 0,C 180,E1 -24249.103,E2 -24249.103} C_VEL
LIN {X 0,Y 159.25,Z 328.099,A -85,B 0,C 180,E1 -24251.016,E2 -24251.016} C_VEL
LIN {X 0,Y 154.234,Z 317.443,A -85,B 0,C 180,E1 -24253.293,E2 -24253.293} C_VEL
LIN {X 0,Y 149.044,Z 307.879,A -85,B 0,C 180,E1 -24255.814,E2 -24255.814} C_VEL
LIN {X 0,Y 146.151,Z 302.919,A -85,B 0,C 180,E1 -24257.325,E2 -24257.325} C_VEL
LIN {X 0,Y 143.69,Z 299.578,A -85,B 0,C 180,E1 -24258.63,E2 -24258.63} C_VEL
LIN {X 0,Y 143.163,Z 297.834,A -85,B 0,C 180,E1 -24259.028,E2 -24259.028} C_VEL
LIN {X 0,Y 143.059,Z 297.482,A -85,B 0,C 180,E1 -24259.654,E2 -24259.654} C_VEL
LIN {X 0,Y 143.083,Z 297.477,A -85,B 0,C 180,E1 -24263.885,E2 -24263.885} C_VEL
LIN {X 0,Y 143.172,Z 297.463,A -85,B 0,C 180,E1 -24267.319,E2 -24267.319} C_VEL
LIN {X 0,Y 143.107,Z 297.474,A -85,B 0,C 180,E1 -24273.769,E2 -24273.769} C_VEL
LIN {X 0,Y 143.248,Z 297.45,A -85,B 0,C 180,E1 -24279.914,E2 -24279.914} C_VEL
LIN {X 0,Y 143.306,Z 297.446,A -85,B 0,C 180,E1 -24285.806,E2 -24285.806} C_VEL
LIN {X 0,Y 143.534,Z 297.404,A -85,B 0,C 180,E1 -24288.706,E2 -24288.706} C_VEL
LIN {X 0,Y 143.607,Z 297.368,A -85,B 0,C 180,E1 -24291.558,E2 -24291.558} C_VEL
LIN {X 0,Y 144.157,Z 297.33,A -85,B 0,C 180,E1 -24300,E2 -24300} C_VEL
LIN {X 0,Y 143.621,Z 297.405,A -85,B 0,C 180,E1 -24308.442,E2 -24308.442} C_VEL
LIN {X 0,Y 143.5,Z 297.412,A -85,B 0,C 180,E1 -24311.613,E2 -24311.613} C_VEL
LIN {X 0,Y 143.251,Z 297.426,A -85,B 0,C 180,E1 -24317.12,E2 -24317.12} C_VEL
LIN {X 0,Y 143.221,Z 297.456,A -85,B 0,C 180,E1 -24321.193,E2 -24321.193} C_VEL
LIN {X 0,Y 143.144,Z 297.459,A -85,B 0,C 180,E1 -24327.899,E2 -24327.899} C_VEL
LIN {X 0,Y 143.141,Z 297.444,A -85,B 0,C 180,E1 -24333.416,E2 -24333.416} C_VEL
LIN {X 0,Y 143.054,Z 297.478,A -85,B 0,C 180,E1 -24339.693,E2 -24339.693} C_VEL
LIN {X 0,Y 143.1,Z 297.624,A -85,B 0,C 180,E1 -24341.783,E2 -24341.783} C_VEL
LIN {X 0,Y 144.003,Z 300.234,A -85,B 0,C 180,E1 -24342.38,E2 -24342.38} C_VEL
LIN {X 0,Y 146.441,Z 302.967,A -85,B 0,C 180,E1 -24343.622,E2 -24343.622} C_VEL
LIN {X 0,Y 148.579,Z 306.285,A -85,B 0,C 180,E1 -24344.718,E2 -24344.718} C_VEL
LIN {X 0,Y 149.97,Z 308.245,A -85,B 0,C 180,E1 -24345.39,E2 -24345.39} C_VEL
LIN {X 0,Y 153.329,Z 313.307,A -85,B 0,C 180,E1 -24346.954,E2 -24346.954} C_VEL
LIN {X 0,Y 158.301,Z 321.287,A -85,B 0,C 180,E1 -24349.109,E2 -24349.109} C_VEL
LIN {X 0,Y 164.475,Z 332.917,A -85,B 0,C 180,E1 -24351.614,E2 -24351.614} C_VEL
LIN {X 0,Y 166.923,Z 338.261,A -85,B 0,C 180,E1 -24352.572,E2 -24352.572} C_VEL
LIN {X 0,Y 165.531,Z 362.837,A -85,B 0,C 180,E1 -24353.601,E2 -24353.601} C_VEL
LIN {X 0,Y 164.598,Z 372.382,A -85,B 0,C 180,E1 -24354.285,E2 -24354.285} C_VEL
LIN {X 0,Y 163.275,Z 382.721,A -85,B 0,C 180,E1 -24355.433,E2 -24355.433} C_VEL
LIN {X 0,Y 161.114,Z 393.004,A -85,B 0,C 180,E1 -24356.956,E2 -24356.956} C_VEL
LIN {X 0,Y 158.37,Z 402.859,A -85,B 0,C 180,E1 -24358.942,E2 -24358.942} C_VEL
LIN {X 0,Y 155.866,Z 410.744,A -85,B 0,C 180,E1 -24361.005,E2 -24361.005} C_VEL
LIN {X 0,Y 154.02,Z 416.392,A -85,B 0,C 180,E1 -24362.85,E2 -24362.85} C_VEL
LIN {X 0,Y 151.535,Z 422.712,A -85,B 0,C 180,E1 -24365.327,E2 -24365.327} C_VEL
LIN {X 0,Y 149.303,Z 427.962,A -85,B 0,C 180,E1 -24367.877,E2 -24367.877} C_VEL
LIN {X 0,Y 147.309,Z 432.344,A -85,B 0,C 180,E1 -24370.489,E2 -24370.489} C_VEL
LIN {X 0,Y 144.912,Z 437.491,A -85,B 0,C 180,E1 -24374.528,E2 -24374.528} C_VEL
LIN {X 0,Y 143.655,Z 440.127,A -85,B 0,C 180,E1 -24377.281,E2 -24377.281} C_VEL
LIN {X 0,Y 142.323,Z 443.009,A -85,B 0,C 180,E1 -24381.479,E2 -24381.479} C_VEL
LIN {X 0,Y 141.689,Z 444.267,A -85,B 0,C 180,E1 -24384.305,E2 -24384.305} C_VEL
LIN {X 0,Y 141.274,Z 445.06,A -85,B 0,C 180,E1 -24387.147,E2 -24387.147} C_VEL
LIN {X 0,Y 141.15,Z 445.361,A -85,B 0,C 180,E1 -24389.999,E2 -24389.999} C_VEL
LIN {X 0,Y 141.27,Z 445.082,A -85,B 0,C 180,E1 -24392.85,E2 -24392.85} C_VEL
LIN {X 0,Y 141.665,Z 444.332,A -85,B 0,C 180,E1 -24395.693,E2 -24395.693} C_VEL
LIN {X 0,Y 142.859,Z 442.105,A -85,B 0,C 180,E1 -24400.291,E2 -24400.291} C_VEL
LIN {X 0,Y 144.239,Z 439.134,A -85,B 0,C 180,E1 -24404.099,E2 -24404.099} C_VEL
LIN {X 0,Y 146.387,Z 434.497,A -85,B 0,C 180,E1 -24408.182,E2 -24408.182} C_VEL
LIN {X 0,Y 148.711,Z 429.445,A -85,B 0,C 180,E1 -24411.484,E2 -24411.484} C_VEL
LIN {X 0,Y 150.856,Z 424.504,A -85,B 0,C 180,E1 -24414.055,E2 -24414.055} C_VEL
LIN {X 0,Y 153.302,Z 418.535,A -85,B 0,C 180,E1 -24416.549,E2 -24416.549} C_VEL
LIN {X 0,Y 155.789,Z 411.278,A -85,B 0,C 180,E1 -24419.008,E2 -24419.008} C_VEL
LIN {X 0,Y 157.978,Z 404.727,A -85,B 0,C 180,E1 -24420.769,E2 -24420.769} C_VEL
LIN {X 0,Y 160.287,Z 396.787,A -85,B 0,C 180,E1 -24422.486,E2 -24422.486} C_VEL
LIN {X 0,Y 162.236,Z 388.578,A -85,B 0,C 180,E1 -24423.898,E2 -24423.898} C_VEL
LIN {X 0,Y 163.79,Z 380.199,A -85,B 0,C 180,E1 -24425.028,E2 -24425.028} C_VEL
LIN {X 0,Y 165.036,Z 370.422,A -85,B 0,C 180,E1 -24426.023,E2 -24426.023} C_VEL
LIN {X 0,Y 165.868,Z 360.685,A -85,B 0,C 180,E1 -24426.666,E2 -24426.666} C_VEL
LIN {X 0,Y 167.027,Z 338.371,A -85,B 0,C 180,E1 -24427.592,E2 -24427.592} C_VEL
LIN {X 0,Y 161.79,Z 327.573,A -85,B 0,C 180,E1 -24429.664,E2 -24429.664} C_VEL
LIN {X 0,Y 155.985,Z 317.45,A -85,B 0,C 180,E1 -24432.095,E2 -24432.095} C_VEL
LIN {X 0,Y 151.085,Z 309.891,A -85,B 0,C 180,E1 -24434.312,E2 -24434.312} C_VEL
LIN {X 0,Y 148.583,Z 306.252,A -85,B 0,C 180,E1 -24435.522,E2 -24435.522} C_VEL
LIN {X 0,Y 146.45,Z 302.977,A -85,B 0,C 180,E1 -24436.619,E2 -24436.619} C_VEL
LIN {X 0,Y 143.849,Z 299.895,A -85,B 0,C 180,E1 -24437.967,E2 -24437.967} C_VEL
LIN {X 0,Y 143.102,Z 297.447,A -85,B 0,C 180,E1 -24438.529,E2 -24438.529} C_VEL
LIN {X 0,Y 143.079,Z 297.466,A -85,B 0,C 180,E1 -24443.882,E2 -24443.882} C_VEL
LIN {X 0,Y 143.169,Z 297.455,A -85,B 0,C 180,E1 -24447.318,E2 -24447.318} C_VEL
LIN {X 0,Y 143.179,Z 297.453,A -85,B 0,C 180,E1 -24452.068,E2 -24452.068} C_VEL
LIN {X 0,Y 143.219,Z 297.455,A -85,B 0,C 180,E1 -24458.802,E2 -24458.802} C_VEL
LIN {X 0,Y 143.247,Z 297.431,A -85,B 0,C 180,E1 -24462.88,E2 -24462.88} C_VEL
LIN {X 0,Y 143.528,Z 297.411,A -85,B 0,C 180,E1 -24468.704,E2 -24468.704} C_VEL
LIN {X 0,Y 143.614,Z 297.406,A -85,B 0,C 180,E1 -24471.558,E2 -24471.558} C_VEL
LIN {X 0,Y 144.15,Z 297.332,A -85,B 0,C 180,E1 -24480,E2 -24480} C_VEL
LIN {X 0,Y 143.615,Z 297.407,A -85,B 0,C 180,E1 -24488.442,E2 -24488.442} C_VEL
LIN {X 0,Y 143.493,Z 297.417,A -85,B 0,C 180,E1 -24491.613,E2 -24491.613} C_VEL
LIN {X 0,Y 143.247,Z 297.453,A -85,B 0,C 180,E1 -24497.12,E2 -24497.12} C_VEL
LIN {X 0,Y 143.214,Z 297.456,A -85,B 0,C 180,E1 -24501.194,E2 -24501.194} C_VEL
LIN {X 0,Y 143.138,Z 297.47,A -85,B 0,C 180,E1 -24507.9,E2 -24507.9} C_VEL
LIN {X 0,Y 143.134,Z 297.472,A -85,B 0,C 180,E1 -24513.417,E2 -24513.417} C_VEL
LIN {X 0,Y 143.048,Z 297.484,A -85,B 0,C 180,E1 -24519.694,E2 -24519.694} C_VEL
LIN {X 0,Y 143.096,Z 297.678,A -85,B 0,C 180,E1 -24520.663,E2 -24520.663} C_VEL
LIN {X 0,Y 143.356,Z 298.657,A -85,B 0,C 180,E1 -24520.987,E2 -24520.987} C_VEL
LIN {X 0,Y 144.69,Z 301.148,A -85,B 0,C 180,E1 -24521.764,E2 -24521.764} C_VEL
LIN {X 0,Y 146.875,Z 304.019,A -85,B 0,C 180,E1 -24522.899,E2 -24522.899} C_VEL
LIN {X 0,Y 150.815,Z 311.158,A -85,B 0,C 180,E1 -24524.938,E2 -24524.938} C_VEL
LIN {X 0,Y 153.487,Z 316.08,A -85,B 0,C 180,E1 -24526.228,E2 -24526.228} C_VEL
LIN {X 0,Y 158.269,Z 325.677,A -85,B 0,C 180,E1 -24528.413,E2 -24528.413} C_VEL
LIN {X 0,Y 163.175,Z 337.958,A -85,B 0,C 180,E1 -24530.591,E2 -24530.591} C_VEL
LIN {X 0,Y 163.811,Z 340.679,A -85,B 0,C 180,E1 -24530.921,E2 -24530.921} C_VEL
LIN {X 0,Y 165.714,Z 362.872,A -85,B 0,C 180,E1 -24532.635,E2 -24532.635} C_VEL
LIN {X 0,Y 164.621,Z 380.682,A -85,B 0,C 180,E1 -24533.45,E2 -24533.45} C_VEL
LIN {X 0,Y 162.895,Z 392.744,A -85,B 0,C 180,E1 -24534.455,E2 -24534.455} C_VEL
LIN {X 0,Y 161.13,Z 401.244,A -85,B 0,C 180,E1 -24535.459,E2 -24535.459} C_VEL
LIN {X 0,Y 158.954,Z 409.918,A -85,B 0,C 180,E1 -24536.83,E2 -24536.83} C_VEL
LIN {X 0,Y 156.548,Z 418.01,A -85,B 0,C 180,E1 -24538.481,E2 -24538.481} C_VEL
LIN {X 0,Y 154.196,Z 425.051,A -85,B 0,C 180,E1 -24540.288,E2 -24540.288} C_VEL
LIN {X 0,Y 151.742,Z 431.724,A -85,B 0,C 180,E1 -24542.411,E2 -24542.411} C_VEL
LIN {X 0,Y 149.155,Z 438.062,A -85,B 0,C 180,E1 -24544.91,E2 -24544.91} C_VEL
LIN {X 0,Y 146.993,Z 443.34,A -85,B 0,C 180,E1 -24547.513,E2 -24547.513} C_VEL
LIN {X 0,Y 145.061,Z 447.741,A -85,B 0,C 180,E1 -24550.177,E2 -24550.177} C_VEL
LIN {X 0,Y 142.902,Z 452.951,A -85,B 0,C 180,E1 -24554.308,E2 -24554.308} C_VEL
LIN {X 0,Y 141.515,Z 456.789,A -85,B 0,C 180,E1 -24558.543,E2 -24558.543} C_VEL
LIN {X 0,Y 140.985,Z 458.559,A -85,B 0,C 180,E1 -24561.401,E2 -24561.401} C_VEL
LIN {X 0,Y 140.749,Z 459.832,A -85,B 0,C 180,E1 -24564.27,E2 -24564.27} C_VEL
LIN {X 0,Y 140.778,Z 460.63,A -85,B 0,C 180,E1 -24567.14,E2 -24567.14} C_VEL
LIN {X 0,Y 141.021,Z 460.941,A -85,B 0,C 180,E1 -24570.001,E2 -24570.001} C_VEL
LIN {X 0,Y 140.777,Z 460.58,A -85,B 0,C 180,E1 -24573.185,E2 -24573.185} C_VEL
LIN {X 0,Y 140.986,Z 458.502,A -85,B 0,C 180,E1 -24578.602,E2 -24578.602} C_VEL
LIN {X 0,Y 141.877,Z 455.536,A -85,B 0,C 180,E1 -24582.882,E2 -24582.882} C_VEL
LIN {X 0,Y 142.898,Z 452.844,A -85,B 0,C 180,E1 -24585.696,E2 -24585.696} C_VEL
LIN {X 0,Y 144.07,Z 449.94,A -85,B 0,C 180,E1 -24588.152,E2 -24588.152} C_VEL
LIN {X 0,Y 144.64,Z 447.171,A -85,B 0,C 180,E1 -24590.213,E2 -24590.213} C_VEL
LIN {X 0,Y 144.138,Z 442.069,A -85,B 0,C 180,E1 -24593.587,E2 -24593.587} C_VEL
LIN {X 0,Y 143.967,Z 436.247,A -85,B 0,C 180,E1 -24596.771,E2 -24596.771} C_VEL
LIN {X 0,Y 145.009,Z 432.247,A -85,B 0,C 180,E1 -24598.457,E2 -24598.457} C_VEL
LIN {X 0,Y 147.745,Z 425.401,A -85,B 0,C 180,E1 -24600.756,E2 -24600.756} C_VEL
LIN {X 0,Y 150.117,Z 418.535,A -85,B 0,C 180,E1 -24602.63,E2 -24602.63} C_VEL
LIN {X 0,Y 152.58,Z 410.595,A -85,B 0,C 180,E1 -24604.352,E2 -24604.352} C_VEL
LIN {X 0,Y 154.826,Z 402.186,A -85,B 0,C 180,E1 -24605.764,E2 -24605.764} C_VEL
LIN {X 0,Y 156.8,Z 393.459,A -85,B 0,C 180,E1 -24606.856,E2 -24606.856} C_VEL
LIN {X 0,Y 158.543,Z 382.904,A -85,B 0,C 180,E1 -24607.805,E2 -24607.805} C_VEL
LIN {X 0,Y 159.7,Z 368.779,A -85,B 0,C 180,E1 -24608.561,E2 -24608.561} C_VEL
LIN {X 0,Y 159.869,Z 362.335,A -85,B 0,C 180,E1 -24608.875,E2 -24608.875} C_VEL
LIN {X 0,Y 158.187,Z 341.753,A -85,B 0,C 180,E1 -24610.548,E2 -24610.548} C_VEL
LIN {X 0,Y 153.456,Z 329.496,A -85,B 0,C 180,E1 -24612.81,E2 -24612.81} C_VEL
LIN {X 0,Y 147.731,Z 317.724,A -85,B 0,C 180,E1 -24615.663,E2 -24615.663} C_VEL
LIN {X 0,Y 142.385,Z 308.071,A -85,B 0,C 180,E1 -24618.587,E2 -24618.587} C_VEL
LIN {X 0,Y 139.897,Z 304.482,A -85,B 0,C 180,E1 -24620.017,E2 -24620.017} C_VEL
LIN {X 0,Y 139.278,Z 303.495,A -85,B 0,C 180,E1 -24620.394,E2 -24620.394} C_VEL
LIN {X 0,Y 137.112,Z 301.345,A -85,B 0,C 180,E1 -24621.661,E2 -24621.661} C_VEL
LIN {X 0,Y 136.09,Z 298.845,A -85,B 0,C 180,E1 -24622.409,E2 -24622.409} C_VEL
LIN {X 0,Y 136.017,Z 298.359,A -85,B 0,C 180,E1 -24622.619,E2 -24622.619} C_VEL
LIN {X 0,Y 136.052,Z 298.353,A -85,B 0,C 180,E1 -24625.744,E2 -24625.744} C_VEL
LIN {X 0,Y 136.085,Z 298.344,A -85,B 0,C 180,E1 -24632.303,E2 -24632.303} C_VEL
LIN {X 0,Y 136.183,Z 298.332,A -85,B 0,C 180,E1 -24638.823,E2 -24638.823} C_VEL
LIN {X 0,Y 136.224,Z 298.326,A -85,B 0,C 180,E1 -24645.051,E2 -24645.051} C_VEL
LIN {X 0,Y 136.428,Z 298.294,A -85,B 0,C 180,E1 -24648.179,E2 -24648.179} C_VEL
LIN {X 0,Y 136.536,Z 298.249,A -85,B 0,C 180,E1 -24651.117,E2 -24651.117} C_VEL
LIN {X 0,Y 137.114,Z 298.206,A -85,B 0,C 180,E1 -24660,E2 -24660} C_VEL
LIN {X 0,Y 136.547,Z 298.288,A -85,B 0,C 180,E1 -24668.883,E2 -24668.883} C_VEL
LIN {X 0,Y 136.416,Z 298.289,A -85,B 0,C 180,E1 -24671.893,E2 -24671.893} C_VEL
LIN {X 0,Y 136.165,Z 298.319,A -85,B 0,C 180,E1 -24678.041,E2 -24678.041} C_VEL
LIN {X 0,Y 136.146,Z 298.335,A -85,B 0,C 180,E1 -24681.689,E2 -24681.689} C_VEL
LIN {X 0,Y 136.065,Z 298.341,A -85,B 0,C 180,E1 -24688.585,E2 -24688.585} C_VEL
LIN {X 0,Y 136.043,Z 298.322,A -85,B 0,C 180,E1 -24694.63,E2 -24694.63} C_VEL
LIN {X 0,Y 136.03,Z 298.353,A -85,B 0,C 180,E1 -24698.315,E2 -24698.315} C_VEL
LIN {X 0,Y 136.914,Z 301.009,A -85,B 0,C 180,E1 -24699.03,E2 -24699.03} C_VEL
LIN {X 0,Y 138.805,Z 303.115,A -85,B 0,C 180,E1 -24700.164,E2 -24700.164} C_VEL
LIN {X 0,Y 139.66,Z 304.075,A -85,B 0,C 180,E1 -24700.659,E2 -24700.659} C_VEL
LIN {X 0,Y 141.807,Z 307.381,A -85,B 0,C 180,E1 -24701.921,E2 -24701.921} C_VEL
LIN {X 0,Y 143.161,Z 309.119,A -85,B 0,C 180,E1 -24702.657,E2 -24702.657} C_VEL
LIN {X 0,Y 148.298,Z 316.624,A -85,B 0,C 180,E1 -24705.306,E2 -24705.306} C_VEL
LIN {X 0,Y 154.227,Z 326.444,A -85,B 0,C 180,E1 -24708.084,E2 -24708.084} C_VEL
LIN {X 0,Y 159.951,Z 337.583,A -85,B 0,C 180,E1 -24710.566,E2 -24710.566} C_VEL
LIN {X 0,Y 161.221,Z 340.367,A -85,B 0,C 180,E1 -24711.099,E2 -24711.099} C_VEL
LIN {X 0,Y 159.863,Z 363.52,A -85,B 0,C 180,E1 -24712.109,E2 -24712.109} C_VEL
LIN {X 0,Y 158.766,Z 373.846,A -85,B 0,C 180,E1 -24712.884,E2 -24712.884} C_VEL
LIN {X 0,Y 156.896,Z 386.123,A -85,B 0,C 180,E1 -24714.384,E2 -24714.384} C_VEL
LIN {X 0,Y 154.833,Z 394.897,A -85,B 0,C 180,E1 -24715.824,E2 -24715.824} C_VEL
LIN {X 0,Y 152.361,Z 403.253,A -85,B 0,C 180,E1 -24717.571,E2 -24717.571} C_VEL
LIN {X 0,Y 149.704,Z 411.139,A -85,B 0,C 180,E1 -24719.689,E2 -24719.689} C_VEL
LIN {X 0,Y 147.745,Z 416.787,A -85,B 0,C 180,E1 -24721.595,E2 -24721.595} C_VEL
LIN {X 0,Y 145.132,Z 423.105,A -85,B 0,C 180,E1 -24724.161,E2 -24724.161} C_VEL
LIN {X 0,Y 142.781,Z 428.354,A -85,B 0,C 180,E1 -24726.809,E2 -24726.809} C_VEL
LIN {X 0,Y 140.642,Z 432.738,A -85,B 0,C 180,E1 -24729.524,E2 -24729.524} C_VEL
LIN {X 0,Y 138.094,Z 437.883,A -85,B 0,C 180,E1 -24733.744,E2 -24733.744} C_VEL
LIN {X 0,Y 136.75,Z 440.519,A -85,B 0,C 180,E1 -24736.627,E2 -24736.627} C_VEL
LIN {X 0,Y 135.315,Z 443.401,A -85,B 0,C 180,E1 -24741.034,E2 -24741.034} C_VEL
LIN {X 0,Y 134.653,Z 444.657,A -85,B 0,C 180,E1 -24744.007,E2 -24744.007} C_VEL
LIN {X 0,Y 134.21,Z 445.451,A -85,B 0,C 180,E1 -24746.997,E2 -24746.997} C_VEL
LIN {X 0,Y 134.075,Z 445.752,A -85,B 0,C 180,E1 -24749.998,E2 -24749.998} C_VEL
LIN {X 0,Y 134.205,Z 445.472,A -85,B 0,C 180,E1 -24753,E2 -24753} C_VEL
LIN {X 0,Y 134.63,Z 444.722,A -85,B 0,C 180,E1 -24755.991,E2 -24755.991} C_VEL
LIN {X 0,Y 135.716,Z 442.787,A -85,B 0,C 180,E1 -24760.29,E2 -24760.29} C_VEL
LIN {X 0,Y 137.391,Z 439.523,A -85,B 0,C 180,E1 -24764.817,E2 -24764.817} C_VEL
LIN {X 0,Y 139.683,Z 434.887,A -85,B 0,C 180,E1 -24769.088,E2 -24769.088} C_VEL
LIN {X 0,Y 142.159,Z 429.833,A -85,B 0,C 180,E1 -24772.527,E2 -24772.527} C_VEL
LIN {X 0,Y 144.422,Z 424.892,A -85,B 0,C 180,E1 -24775.2,E2 -24775.2} C_VEL
LIN {X 0,Y 147.007,Z 418.922,A -85,B 0,C 180,E1 -24777.781,E2 -24777.781} C_VEL
LIN {X 0,Y 149.647,Z 411.665,A -85,B 0,C 180,E1 -24780.32,E2 -24780.32} C_VEL
LIN {X 0,Y 151.948,Z 405.113,A -85,B 0,C 180,E1 -24782.133,E2 -24782.133} C_VEL
LIN {X 0,Y 154.368,Z 397.173,A -85,B 0,C 180,E1 -24783.896,E2 -24783.896} C_VEL
LIN {X 0,Y 156.411,Z 388.963,A -85,B 0,C 180,E1 -24785.344,E2 -24785.344} C_VEL
LIN {X 0,Y 157.978,Z 380.956,A -85,B 0,C 180,E1 -24786.458,E2 -24786.458} C_VEL
LIN {X 0,Y 159.286,Z 371.329,A -85,B 0,C 180,E1 -24787.478,E2 -24787.478} C_VEL
LIN {X 0,Y 160.206,Z 361.675,A -85,B 0,C 180,E1 -24788.141,E2 -24788.141} C_VEL
LIN {X 0,Y 161.372,Z 340.578,A -85,B 0,C 180,E1 -24789.051,E2 -24789.051} C_VEL
LIN {X 0,Y 156.254,Z 330.114,A -85,B 0,C 180,E1 -24791.238,E2 -24791.238} C_VEL
LIN {X 0,Y 150.1,Z 319.414,A -85,B 0,C 180,E1 -24794.057,E2 -24794.057} C_VEL
LIN {X 0,Y 145.019,Z 311.761,A -85,B 0,C 180,E1 -24796.6,E2 -24796.6} C_VEL
LIN {X 0,Y 142.116,Z 307.638,A -85,B 0,C 180,E1 -24798.177,E2 -24798.177} C_VEL
LIN {X 0,Y 139.833,Z 304.373,A -85,B 0,C 180,E1 -24799.501,E2 -24799.501} C_VEL
LIN {X 0,Y 139.103,Z 303.359,A -85,B 0,C 180,E1 -24799.939,E2 -24799.939} C_VEL
LIN {X 0,Y 136.994,Z 301.163,A -85,B 0,C 180,E1 -24801.195,E2 -24801.195} C_VEL
LIN {X 0,Y 136.134,Z 298.981,A -85,B 0,C 180,E1 -24801.837,E2 -24801.837} C_VEL
LIN {X 0,Y 136.036,Z 298.348,A -85,B 0,C 180,E1 -24802.04,E2 -24802.04} C_VEL
LIN {X 0,Y 136.048,Z 298.348,A -85,B 0,C 180,E1 -24805.741,E2 -24805.741} C_VEL
LIN {X 0,Y 136.12,Z 298.332,A -85,B 0,C 180,E1 -24812.31,E2 -24812.31} C_VEL
LIN {X 0,Y 136.182,Z 298.331,A -85,B 0,C 180,E1 -24818.823,E2 -24818.823} C_VEL
LIN {X 0,Y 136.218,Z 298.291,A -85,B 0,C 180,E1 -24825.05,E2 -24825.05} C_VEL
LIN {X 0,Y 136.421,Z 298.287,A -85,B 0,C 180,E1 -24828.178,E2 -24828.178} C_VEL
LIN {X 0,Y 136.54,Z 298.289,A -85,B 0,C 180,E1 -24831.117,E2 -24831.117} C_VEL
LIN {X 0,Y 137.107,Z 298.208,A -85,B 0,C 180,E1 -24840,E2 -24840} C_VEL
LIN {X 0,Y 136.541,Z 298.286,A -85,B 0,C 180,E1 -24848.883,E2 -24848.883} C_VEL
LIN {X 0,Y 136.409,Z 298.301,A -85,B 0,C 180,E1 -24851.893,E2 -24851.893} C_VEL
LIN {X 0,Y 136.16,Z 298.339,A -85,B 0,C 180,E1 -24858.04,E2 -24858.04} C_VEL
LIN {X 0,Y 136.139,Z 298.339,A -85,B 0,C 180,E1 -24861.69,E2 -24861.69} C_VEL
LIN {X 0,Y 136.058,Z 298.353,A -85,B 0,C 180,E1 -24868.586,E2 -24868.586} C_VEL
LIN {X 0,Y 136.036,Z 298.357,A -85,B 0,C 180,E1 -24874.631,E2 -24874.631} C_VEL
LIN {X 0,Y 136.005,Z 298.36,A -85,B 0,C 180,E1 -24877.269,E2 -24877.269} C_VEL
LIN {X 0,Y 136.993,Z 301.164,A -85,B 0,C 180,E1 -24878.073,E2 -24878.073} C_VEL
LIN {X 0,Y 139.04,Z 303.321,A -85,B 0,C 180,E1 -24879.295,E2 -24879.295} C_VEL
LIN {X 0,Y 139.776,Z 304.254,A -85,B 0,C 180,E1 -24879.73,E2 -24879.73} C_VEL
LIN {X 0,Y 142.014,Z 307.55,A -85,B 0,C 180,E1 -24881.039,E2 -24881.039} C_VEL
LIN {X 0,Y 145.79,Z 314.031,A -85,B 0,C 180,E1 -24883.151,E2 -24883.151} C_VEL
LIN {X 0,Y 151.59,Z 325.364,A -85,B 0,C 180,E1 -24886.143,E2 -24886.143} C_VEL
LIN {X 0,Y 156.611,Z 337.195,A -85,B 0,C 180,E1 -24888.57,E2 -24888.57} C_VEL
LIN {X 0,Y 158.398,Z 342.652,A -85,B 0,C 180,E1 -24889.448,E2 -24889.448} C_VEL
LIN {X 0,Y 160.078,Z 363.869,A -85,B 0,C 180,E1 -24891.156,E2 -24891.156} C_VEL
LIN {X 0,Y 159.019,Z 379.668,A -85,B 0,C 180,E1 -24891.889,E2 -24891.889} C_VEL
LIN {X 0,Y 157.299,Z 391.69,A -85,B 0,C 180,E1 -24892.874,E2 -24892.874} C_VEL
LIN {X 0,Y 155.348,Z 400.859,A -85,B 0,C 180,E1 -24893.978,E2 -24893.978} C_VEL
LIN {X 0,Y 153.063,Z 409.531,A -85,B 0,C 180,E1 -24895.377,E2 -24895.377} C_VEL
LIN {X 0,Y 150.814,Z 416.839,A -85,B 0,C 180,E1 -24896.882,E2 -24896.882} C_VEL
LIN {X 0,Y 148.053,Z 424.661,A -85,B 0,C 180,E1 -24898.922,E2 -24898.922} C_VEL
LIN {X 0,Y 145.478,Z 431.334,A -85,B 0,C 180,E1 -24901.114,E2 -24901.114} C_VEL
LIN {X 0,Y 142.736,Z 437.671,A -85,B 0,C 180,E1 -24903.697,E2 -24903.697} C_VEL
LIN {X 0,Y 140.458,Z 442.949,A -85,B 0,C 180,E1 -24906.405,E2 -24906.405} C_VEL
LIN {X 0,Y 138.399,Z 447.351,A -85,B 0,C 180,E1 -24909.18,E2 -24909.18} C_VEL
LIN {X 0,Y 136.061,Z 452.559,A -85,B 0,C 180,E1 -24913.497,E2 -24913.497} C_VEL
LIN {X 0,Y 134.537,Z 456.397,A -85,B 0,C 180,E1 -24917.941,E2 -24917.941} C_VEL
